// TIA Portal V20 export
// export: Created 2025-12-01T14:57:42.2360027Z, ExportSetting None, DisplayName Totally Integrated Automation Portal, DisplayVersion V20 Update 3, DisplayName TIA Portal Openness, DisplayVersion V20 Update 3, DisplayName TIA Portal Version Control Interface, DisplayVersion V20 Update 3, DisplayName STEP 7 Professional, DisplayVersion V20 Update 3, DisplayName STEP 7 Safety, DisplayVersion V20 Update 2, DisplayName WinCC Basic/Comfort/Advanced, DisplayVersion V20 Update 3, DisplayName WinCC Professional, DisplayVersion V20 Update 3, DisplayName WinCC Unified, DisplayVersion V20 Update 3
FUNCTION_BLOCK "FB383_GarrasLenze_Paletizador_NDD_E3S3"   // FB383, LAD
{ S7_Optimized_Access := 'FALSE' }
// stored: AutoNumber false, SetENOAutomatically false
   VAR_INPUT
      Mesa : UInt;   // Mesa de la FB
      NDB_ConfigNDD : UInt;
      NDB_DatosNDD : UInt;   // DB de Configuracion Particular del NDD
      OffsetDatosGarra : UInt;
      DesHabilitar_Garra : Bool;
      Mantenimiento : Bool;
      Error_Tx : Bool;
      EnTension : Bool;   // Existe Tension en la Mesa
      TermicoFRENO_Garra : Bool;
      Garra_PresCarga : Bool;
      EM_Garra_Down : Bool;
      Garra_Down : Bool;
      Garra_FinPaletizado : Bool;
      Garra_InicioPaletizado : Bool;
      EM_Garra_Up : Bool;
      P_Puesto_Capa : Bool;
      P_Puesto_Subir : Bool;
      P_Puesto_Bajar : Bool;
      BarreraNivel : Bool;
      F_EnvMens_PMx : Bool;
      Manual_GarraUp : Bool;
      Manual_GarraDown : Bool;
      Homming_Garra : Bool;   // Realizar el Homing del Variador de la Horquilla (RefCero >> Out)
      pHsRef_Garra : Bool;
      V_TOut_MovGarra : Time;
   END_VAR
   VAR_OUTPUT
      P_EnvMens_PMx : Bool;
   END_VAR
   VAR_IN_OUT
      Interlock_Garras : "NDD_Interlock_Garras";
   END_VAR
   VAR
      TOut_MovGarras { S7_SetPoint := 'True'} : TON_TIME;
      TEstableMovGarras { S7_SetPoint := 'True'} : TON_TIME;
      TEsperaMoverGarras { S7_SetPoint := 'True'} : TON_TIME;
      MemoAlturaPedido : Int;
      MemoEventoPaletizado : UInt;
      MemoPosicionAcutual_Garras : Int;
      PosicionActual_Garras : Int;
      PosicionUp_Garras : Int;
      PosicionDown_Garras : Int;
      PosicionMover_Garras : Int;
      ConsignaFR_Garras : Int;
      SubjectArea_Garras : Word;
      IDArea_Garras : Word;
      NodoNoPres_VarGarras : Bool;   // Nodo del Variador de la Horquilla - No presente
      MoverGarras : Bool;
      FinMoverGarras : Bool;
      MemoFinMoverGarras : Bool;
      PosGarrasUp_OK : Bool;
      PosGarrasDown_OK : Bool;
      PosGarrasTransfer_OK : Bool;
      Memo_NuevaCapa : Bool;
      MA_Puesto_NuevaCapa : Bool;
      MA_Puesto_Subir : Bool;
      MA_Puesto_Bajar : Bool;
      MA_Puesto_Baliza : Bool;
      MA_Garras_Subir : Bool;
      MA_Garras_Bajar : Bool;
      GARRA_ET00 : Bool;
      GARRA_ET01 : Bool;
      GARRA_ET02 : Bool;
      GARRA_RST01 : Bool;
      GARRA_RST02 : Bool;
      GARRA_CAR01 : Bool;
      GARRA_CAR02 : Bool;
      GARRA_CAR03 : Bool;
      GARRA_CAR04 : Bool;
      GARRA_DCAR01 : Bool;
      GARRA_DCAR02 : Bool;
      GARRA_DCAR03 : Bool;
      GARRA_DCAR04 : Bool;
      STAT_P_EnvMens_PMx : Bool;
      MemoReferenciaOK_Garra : Bool;
      ErrorVar_Garra : Bool;
      ReferenciaOK_Garra : Bool;
      MemoHoming_Garra : Bool;
      EventoInicioPaletizado : Bool;
      EventoFinalPaletizado : Bool;
      EventoAlturaPedido : Bool;
   END_VAR
   VAR_TEMP
      EstadoZona : "EstadoZona";
      EstadoVI : "EstadosMesa_GarrasLenze_Paletizador_NDD";
      NodoVar_Garra : "Status_NodosProfinet";
      Guardar_AR1 : DWord;
      Guardar_AR2 : DWord;
      P_DatosGarras : DWord;
      P_NodoVar_Garras : DWord;
      DB_ConfigNDD : Word;
      DB_DatosNDD : Word;
      NumDB_DiagProfinet : Word;
      NumNodo_VarGarras : UInt;
      ByteInicial_VarGarras : UInt;
      VeloManual_Garras : Int;
      VeloPuesto_Garras : Int;
      VeloLentaUp_Garras : Int;
      VeloRapidaUp_Garras : Int;
      PosLentaUp_Garras : Int;
      VeloLentaDown_Garras : Int;
      VeloRapidaDown_Garras : Int;
      PosLentaDown_Garras : Int;
      AuxMargen : Int;
      AuxPosMax : Int;
      AuxPosMin : Int;
      AuxAlturaPedidoMax : Int;
      AuxAlturaPedidoMin : Int;
      MargenPedido : Int;
      TempInt : Int;
      AuxEstados : Bool;
      DestinoGarra_DOWN : Bool;
      DestinoGarra_UP : Bool;
      MoverGarra_LentaDOWN : Bool;
      MoverGarra_LentaUP : Bool;
      CalcularAlturaPedido : Bool;
   END_VAR
   VAR_TEMP   // added for the SCL form of the ladder/FBD networks
      _w1 : Bool;
      _w2 : Bool;
      _w3 : Bool;
   END_VAR
BEGIN

REGION Network 1: Inicializaciones
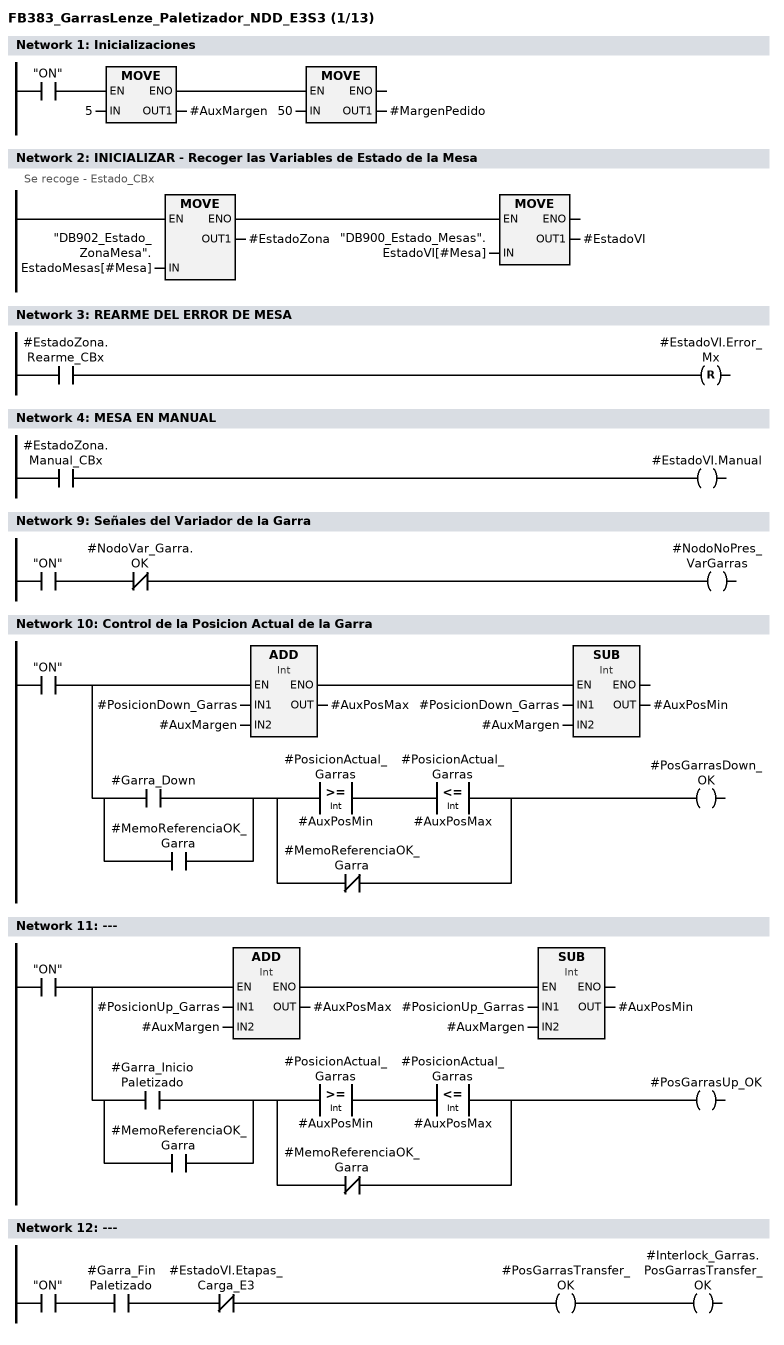
   RUNG wire#powerrail
      Contact( "ON" )
      { S7_GenerateENO := "TRUE" } Move(in := 5, out1 => #AuxMargen)
      { S7_GenerateENO := "TRUE" } Move(in := 50, out1 => #MargenPedido)
   END_RUNG
   // the same network as SCL:
   // ENO of a box is taken as its EN; it also drops when the box reports an error
   IF "ON" THEN
       #AuxMargen := 5;
       #MargenPedido := 50;
   END_IF;
END_REGION

REGION Network 2: INICIALIZAR - Recoger las Variables de Estado de la Mesa
   // Se recoge - Estado_CBx
   RUNG wire#powerrail
      Move(in := "DB902_Estado_ZonaMesa".EstadoMesas[#Mesa], out1 => #EstadoZona)
      Move(in := "DB900_Estado_Mesas".EstadoVI[#Mesa], out1 => #EstadoVI)
   END_RUNG
   // the same network as SCL:
   #EstadoZona := "DB902_Estado_ZonaMesa".EstadoMesas[#Mesa];
   #EstadoVI := "DB900_Estado_Mesas".EstadoVI[#Mesa];
END_REGION

REGION Network 3: REARME DEL ERROR DE MESA
   RUNG wire#powerrail
      Contact( #EstadoZona.Rearme_CBx )
      R_Coil( #EstadoVI.Error_Mx )
   END_RUNG
   // the same network as SCL:
   IF #EstadoZona.Rearme_CBx THEN #EstadoVI.Error_Mx := FALSE; END_IF;
END_REGION

REGION Network 4: MESA EN MANUAL
   RUNG wire#powerrail
      Contact( #EstadoZona.Manual_CBx )
      Coil( #EstadoVI.Manual )
   END_RUNG
   // the same network as SCL:
   #EstadoVI.Manual := #EstadoZona.Manual_CBx;
END_REGION

NETWORK
TITLE = Datos Internos de la Garra
// ------------------------------------------------------------------------------------
// ------------------------------------------------------------------------------------
// --- Previas

      TAR1  #Guardar_AR1;  // Guardar AR1 y AR2


// ------------------------------------------------------------------------------------
// ------------------------------------------------------------------------------------
// --- Datos iniciales

      L     #NDB_ConfigNDD;  // - DB del Config de los Paletizadores MDD
      T     #DB_ConfigNDD;  //
      L     #NDB_DatosNDD;  // - DB del Config de los Paletizadores MDD
      T     #DB_DatosNDD;

      L     #OffsetDatosGarra;  //   Puntero a los Datos de Garra
      SLD   3;
      T     #P_DatosGarras;


/////////////////////////////////////////////////////////////////////////////
/////////////////////////////////////////////////////////////////////////////
// --- Sistema de Profinet

      LAR1  P#0.0;  // - Leer Datos de los Variadores
      OPN   DB [#DB_DatosNDD];  //   del NDD

      L     DBW [AR1, P#0.0];  // - Num DB de Profinet
      T     #NumDB_DiagProfinet;
      L     DBW [AR1, P#8.0];  // - Nodos de los Variadores
      T     #NumNodo_VarGarras;
      L     DBW [AR1, P#14.0];  // - Direcciones de los Variadores
      T     #ByteInicial_VarGarras;

      L     P##NodoVar_Garra;  // Puntero del Estado del Nodo del Variador de Garra (TEMPORAL)
      T     #P_NodoVar_Garras;



NETWORK
TITLE = ----
// ------------------------------------------------------------------------------------
// ------------------------------------------------------------------------------------
// --- Datos Generales de Configuracion de los NDD

      LAR1  P#0.0;  // - Leer Datos de Velocidad de la Garra
      OPN   DB [#DB_ConfigNDD];

      L     DBW [AR1, P#30.0];  // - Velocidad en Manual
      T     #VeloManual_Garras;
      L     DBW [AR1, P#32.0];  // - Velocidad en el Puesto
      T     #VeloPuesto_Garras;

      L     DBW [AR1, P#34.0];  // - Velocidad en Auto Up
      T     #VeloLentaUp_Garras;
      L     DBW [AR1, P#36.0];
      T     #VeloRapidaUp_Garras;

      L     DBW [AR1, P#38.0];  // - Velocidad en Auto Down
      T     #VeloLentaDown_Garras;
      L     DBW [AR1, P#40.0];
      T     #VeloRapidaDown_Garras;

      L     DBW [AR1, P#42.0];  // - Posiciones para Cambio de Velocidad
      T     #PosLentaUp_Garras;
      L     DBW [AR1, P#44.0];
      T     #PosLentaDown_Garras;



NETWORK
TITLE = ----
// ------------------------------------------------------------------------------------
// ------------------------------------------------------------------------------------
// --- Datos Particulares de la Garra del NDD

      LAR1  #P_DatosGarras;  // - Leer Datos de la Garra
      OPN   DB [#DB_DatosNDD];
      L     DBD [AR1, P#0.0];
      T     #PosicionUp_Garras;
      L     DBD [AR1, P#4.0];
      T     #PosicionDown_Garras;


// ------------------------------------------------------------------------------------
// ------------------------------------------------------------------------------------
// --- Estado del Nodo de PROFINET del Variador de la Garra (DANFFOS)

      L     #NumNodo_VarGarras;  // Nodo de Profinet
      L     1;
      -I;
      L     2;  // Longitud registro datos
      *I;
      SLD   3;
      LAR1;

      OPN   DB [#NumDB_DiagProfinet];  // Leer estado del Nodo de PROFINET
      L     DBW [AR1, P#0.0];
      T     LW [#P_NodoVar_Garras];



NETWORK
TITLE = ---
// ------------------------------------------------------------------------------------
// ------------------------------------------------------------------------------------
// --- Final de Datos Inicialies

      LAR1  #Guardar_AR1;  // Recuperar AR1 y AR2



REGION Network 9: Señales del Variador de la Garra
   RUNG wire#powerrail
      Contact( "ON" )
      I_Contact( #NodoVar_Garra.OK )
      Coil( #NodoNoPres_VarGarras )
   END_RUNG
   // the same network as SCL:
   #NodoNoPres_VarGarras := "ON" AND NOT #NodoVar_Garra.OK;
END_REGION

REGION Network 10: Control de la Posicion Actual de la Garra
   RUNG wire#powerrail
      Contact( "ON" )
      wire#w1
      { S7_Templates := "SrcType := Int"; S7_GenerateENO := "TRUE" } Add(in1 := #PosicionDown_Garras, in2 := #AuxMargen, out => #AuxPosMax)
      { S7_Templates := "SrcType := Int"; S7_GenerateENO := "TRUE" } Sub(in1 := #PosicionDown_Garras, in2 := #AuxMargen, out => #AuxPosMin)
   END_RUNG
   RUNG wire#w1
      Contact( #Garra_Down )
      wire#w2
      { S7_Templates := "SrcType := Int" } GE_Contact(in1 := #PosicionActual_Garras, in2 := #AuxPosMin)
      { S7_Templates := "SrcType := Int" } LE_Contact(in1 := #PosicionActual_Garras, in2 := #AuxPosMax)
      wire#w3
      Coil( #PosGarrasDown_OK )
   END_RUNG
   RUNG wire#w1
      Contact( #MemoReferenciaOK_Garra )
   END_RUNG wire#w2
   RUNG wire#w2
      I_Contact( #MemoReferenciaOK_Garra )
   END_RUNG wire#w3
   // the same network as SCL:
   // ENO of a box is taken as its EN; it also drops when the box reports an error
   IF "ON" THEN
       #AuxPosMax := #PosicionDown_Garras + #AuxMargen;
       #AuxPosMin := #PosicionDown_Garras - #AuxMargen;
   END_IF;
   #PosGarrasDown_OK := "ON" AND (#Garra_Down OR #MemoReferenciaOK_Garra) AND (((#PosicionActual_Garras >= #AuxPosMin) AND (#PosicionActual_Garras <= #AuxPosMax)) OR NOT #MemoReferenciaOK_Garra);
END_REGION

REGION Network 11: ---
   RUNG wire#powerrail
      Contact( "ON" )
      wire#w1
      { S7_Templates := "SrcType := Int"; S7_GenerateENO := "TRUE" } Add(in1 := #PosicionUp_Garras, in2 := #AuxMargen, out => #AuxPosMax)
      { S7_Templates := "SrcType := Int"; S7_GenerateENO := "TRUE" } Sub(in1 := #PosicionUp_Garras, in2 := #AuxMargen, out => #AuxPosMin)
   END_RUNG
   RUNG wire#w1
      Contact( #Garra_InicioPaletizado )
      wire#w2
      { S7_Templates := "SrcType := Int" } GE_Contact(in1 := #PosicionActual_Garras, in2 := #AuxPosMin)
      { S7_Templates := "SrcType := Int" } LE_Contact(in1 := #PosicionActual_Garras, in2 := #AuxPosMax)
      wire#w3
      Coil( #PosGarrasUp_OK )
   END_RUNG
   RUNG wire#w1
      Contact( #MemoReferenciaOK_Garra )
   END_RUNG wire#w2
   RUNG wire#w2
      I_Contact( #MemoReferenciaOK_Garra )
   END_RUNG wire#w3
   // the same network as SCL:
   // ENO of a box is taken as its EN; it also drops when the box reports an error
   IF "ON" THEN
       #AuxPosMax := #PosicionUp_Garras + #AuxMargen;
       #AuxPosMin := #PosicionUp_Garras - #AuxMargen;
   END_IF;
   #PosGarrasUp_OK := "ON" AND (#Garra_InicioPaletizado OR #MemoReferenciaOK_Garra) AND (((#PosicionActual_Garras >= #AuxPosMin) AND (#PosicionActual_Garras <= #AuxPosMax)) OR NOT #MemoReferenciaOK_Garra);
END_REGION

REGION Network 12: ---
   RUNG wire#powerrail
      Contact( "ON" )
      Contact( #Garra_FinPaletizado )
      I_Contact( #EstadoVI.Etapas_Carga_E3 )
      Coil( #PosGarrasTransfer_OK )
      Coil( #Interlock_Garras.PosGarrasTransfer_OK )
   END_RUNG
   // the same network as SCL:
   #PosGarrasTransfer_OK := "ON" AND #Garra_FinPaletizado AND NOT #EstadoVI.Etapas_Carga_E3;
   #Interlock_Garras.PosGarrasTransfer_OK := #PosGarrasTransfer_OK;
END_REGION

REGION Network 13: ----
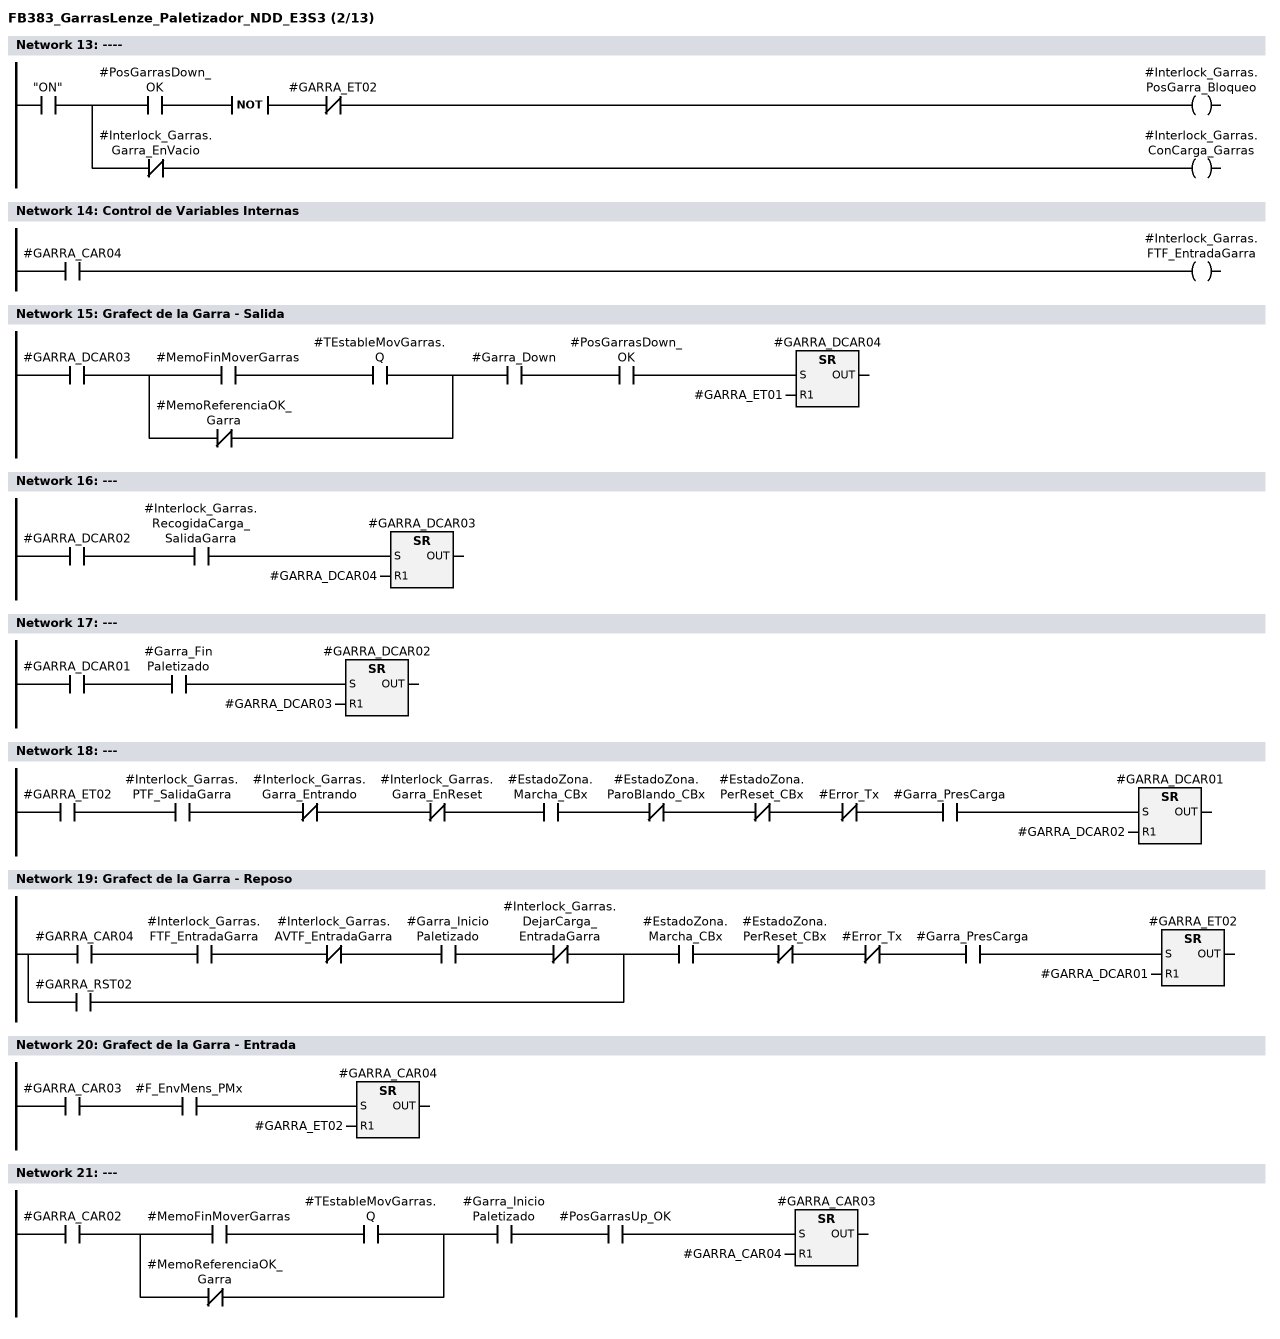
   RUNG wire#powerrail
      Contact( "ON" )
      wire#w1
      Contact( #PosGarrasDown_OK )
      Not()
      I_Contact( #GARRA_ET02 )
      Coil( #Interlock_Garras.PosGarra_Bloqueo )
   END_RUNG
   RUNG wire#w1
      I_Contact( #Interlock_Garras.Garra_EnVacio )
      Coil( #Interlock_Garras.ConCarga_Garras )
   END_RUNG
   // the same network as SCL:
   #Interlock_Garras.PosGarra_Bloqueo := NOT ("ON" AND #PosGarrasDown_OK) AND NOT #GARRA_ET02;
   #Interlock_Garras.ConCarga_Garras := "ON" AND NOT #Interlock_Garras.Garra_EnVacio;
END_REGION

REGION Network 14: Control de Variables Internas
   RUNG wire#powerrail
      Contact( #GARRA_CAR04 )
      Coil( #Interlock_Garras.FTF_EntradaGarra )
   END_RUNG
   // the same network as SCL:
   #Interlock_Garras.FTF_EntradaGarra := #GARRA_CAR04;
END_REGION

REGION Network 15: Grafect de la Garra - Salida
   RUNG wire#powerrail
      Contact( #GARRA_DCAR03 )
      wire#w1
      Contact( #MemoFinMoverGarras )
      Contact( #TEstableMovGarras.Q )
      wire#w2
      Contact( #Garra_Down )
      Contact( #PosGarrasDown_OK )
      S_SR(operand := #GARRA_DCAR04, r1 := #GARRA_ET01)
   END_RUNG
   RUNG wire#w1
      I_Contact( #MemoReferenciaOK_Garra )
   END_RUNG wire#w2
   // the same network as SCL:
   IF #GARRA_DCAR03 AND ((#MemoFinMoverGarras AND #TEstableMovGarras.Q) OR NOT #MemoReferenciaOK_Garra) AND #Garra_Down AND #PosGarrasDown_OK THEN
       #GARRA_DCAR04 := TRUE;   // SR flip-flop
   END_IF;
   IF #GARRA_ET01 THEN #GARRA_DCAR04 := FALSE; END_IF;
END_REGION

REGION Network 16: ---
   RUNG wire#powerrail
      Contact( #GARRA_DCAR02 )
      Contact( #Interlock_Garras.RecogidaCarga_SalidaGarra )
      S_SR(operand := #GARRA_DCAR03, r1 := #GARRA_DCAR04)
   END_RUNG
   // the same network as SCL:
   IF #GARRA_DCAR02 AND #Interlock_Garras.RecogidaCarga_SalidaGarra THEN
       #GARRA_DCAR03 := TRUE;   // SR flip-flop
   END_IF;
   IF #GARRA_DCAR04 THEN #GARRA_DCAR03 := FALSE; END_IF;
END_REGION

REGION Network 17: ---
   RUNG wire#powerrail
      Contact( #GARRA_DCAR01 )
      Contact( #Garra_FinPaletizado )
      S_SR(operand := #GARRA_DCAR02, r1 := #GARRA_DCAR03)
   END_RUNG
   // the same network as SCL:
   IF #GARRA_DCAR01 AND #Garra_FinPaletizado THEN
       #GARRA_DCAR02 := TRUE;   // SR flip-flop
   END_IF;
   IF #GARRA_DCAR03 THEN #GARRA_DCAR02 := FALSE; END_IF;
END_REGION

REGION Network 18: ---
   RUNG wire#powerrail
      Contact( #GARRA_ET02 )
      Contact( #Interlock_Garras.PTF_SalidaGarra )
      I_Contact( #Interlock_Garras.Garra_Entrando )
      I_Contact( #Interlock_Garras.Garra_EnReset )
      Contact( #EstadoZona.Marcha_CBx )
      I_Contact( #EstadoZona.ParoBlando_CBx )
      I_Contact( #EstadoZona.PerReset_CBx )
      I_Contact( #Error_Tx )
      Contact( #Garra_PresCarga )
      S_SR(operand := #GARRA_DCAR01, r1 := #GARRA_DCAR02)
   END_RUNG
   // the same network as SCL:
   IF #GARRA_ET02 AND #Interlock_Garras.PTF_SalidaGarra AND NOT #Interlock_Garras.Garra_Entrando AND NOT #Interlock_Garras.Garra_EnReset AND #EstadoZona.Marcha_CBx AND NOT #EstadoZona.ParoBlando_CBx AND NOT #EstadoZona.PerReset_CBx AND NOT #Error_Tx AND #Garra_PresCarga THEN
       #GARRA_DCAR01 := TRUE;   // SR flip-flop
   END_IF;
   IF #GARRA_DCAR02 THEN #GARRA_DCAR01 := FALSE; END_IF;
END_REGION

REGION Network 19: Grafect de la Garra - Reposo
   RUNG wire#powerrail
      Contact( #GARRA_CAR04 )
      Contact( #Interlock_Garras.FTF_EntradaGarra )
      I_Contact( #Interlock_Garras.AVTF_EntradaGarra )
      Contact( #Garra_InicioPaletizado )
      I_Contact( #Interlock_Garras.DejarCarga_EntradaGarra )
      wire#w1
      Contact( #EstadoZona.Marcha_CBx )
      I_Contact( #EstadoZona.PerReset_CBx )
      I_Contact( #Error_Tx )
      Contact( #Garra_PresCarga )
      S_SR(operand := #GARRA_ET02, r1 := #GARRA_DCAR01)
   END_RUNG
   RUNG wire#powerrail
      Contact( #GARRA_RST02 )
   END_RUNG wire#w1
   // the same network as SCL:
   IF ((#GARRA_CAR04 AND #Interlock_Garras.FTF_EntradaGarra AND NOT #Interlock_Garras.AVTF_EntradaGarra AND #Garra_InicioPaletizado AND NOT #Interlock_Garras.DejarCarga_EntradaGarra) OR #GARRA_RST02) AND #EstadoZona.Marcha_CBx AND NOT #EstadoZona.PerReset_CBx AND NOT #Error_Tx AND #Garra_PresCarga THEN
       #GARRA_ET02 := TRUE;   // SR flip-flop
   END_IF;
   IF #GARRA_DCAR01 THEN #GARRA_ET02 := FALSE; END_IF;
END_REGION

REGION Network 20: Grafect de la Garra - Entrada
   RUNG wire#powerrail
      Contact( #GARRA_CAR03 )
      Contact( #F_EnvMens_PMx )
      S_SR(operand := #GARRA_CAR04, r1 := #GARRA_ET02)
   END_RUNG
   // the same network as SCL:
   IF #GARRA_CAR03 AND #F_EnvMens_PMx THEN
       #GARRA_CAR04 := TRUE;   // SR flip-flop
   END_IF;
   IF #GARRA_ET02 THEN #GARRA_CAR04 := FALSE; END_IF;
END_REGION

REGION Network 21: ---
   RUNG wire#powerrail
      Contact( #GARRA_CAR02 )
      wire#w1
      Contact( #MemoFinMoverGarras )
      Contact( #TEstableMovGarras.Q )
      wire#w2
      Contact( #Garra_InicioPaletizado )
      Contact( #PosGarrasUp_OK )
      S_SR(operand := #GARRA_CAR03, r1 := #GARRA_CAR04)
   END_RUNG
   RUNG wire#w1
      I_Contact( #MemoReferenciaOK_Garra )
   END_RUNG wire#w2
   // the same network as SCL:
   IF #GARRA_CAR02 AND ((#MemoFinMoverGarras AND #TEstableMovGarras.Q) OR NOT #MemoReferenciaOK_Garra) AND #Garra_InicioPaletizado AND #PosGarrasUp_OK THEN
       #GARRA_CAR03 := TRUE;   // SR flip-flop
   END_IF;
   IF #GARRA_CAR04 THEN #GARRA_CAR03 := FALSE; END_IF;
END_REGION

REGION Network 22: ---
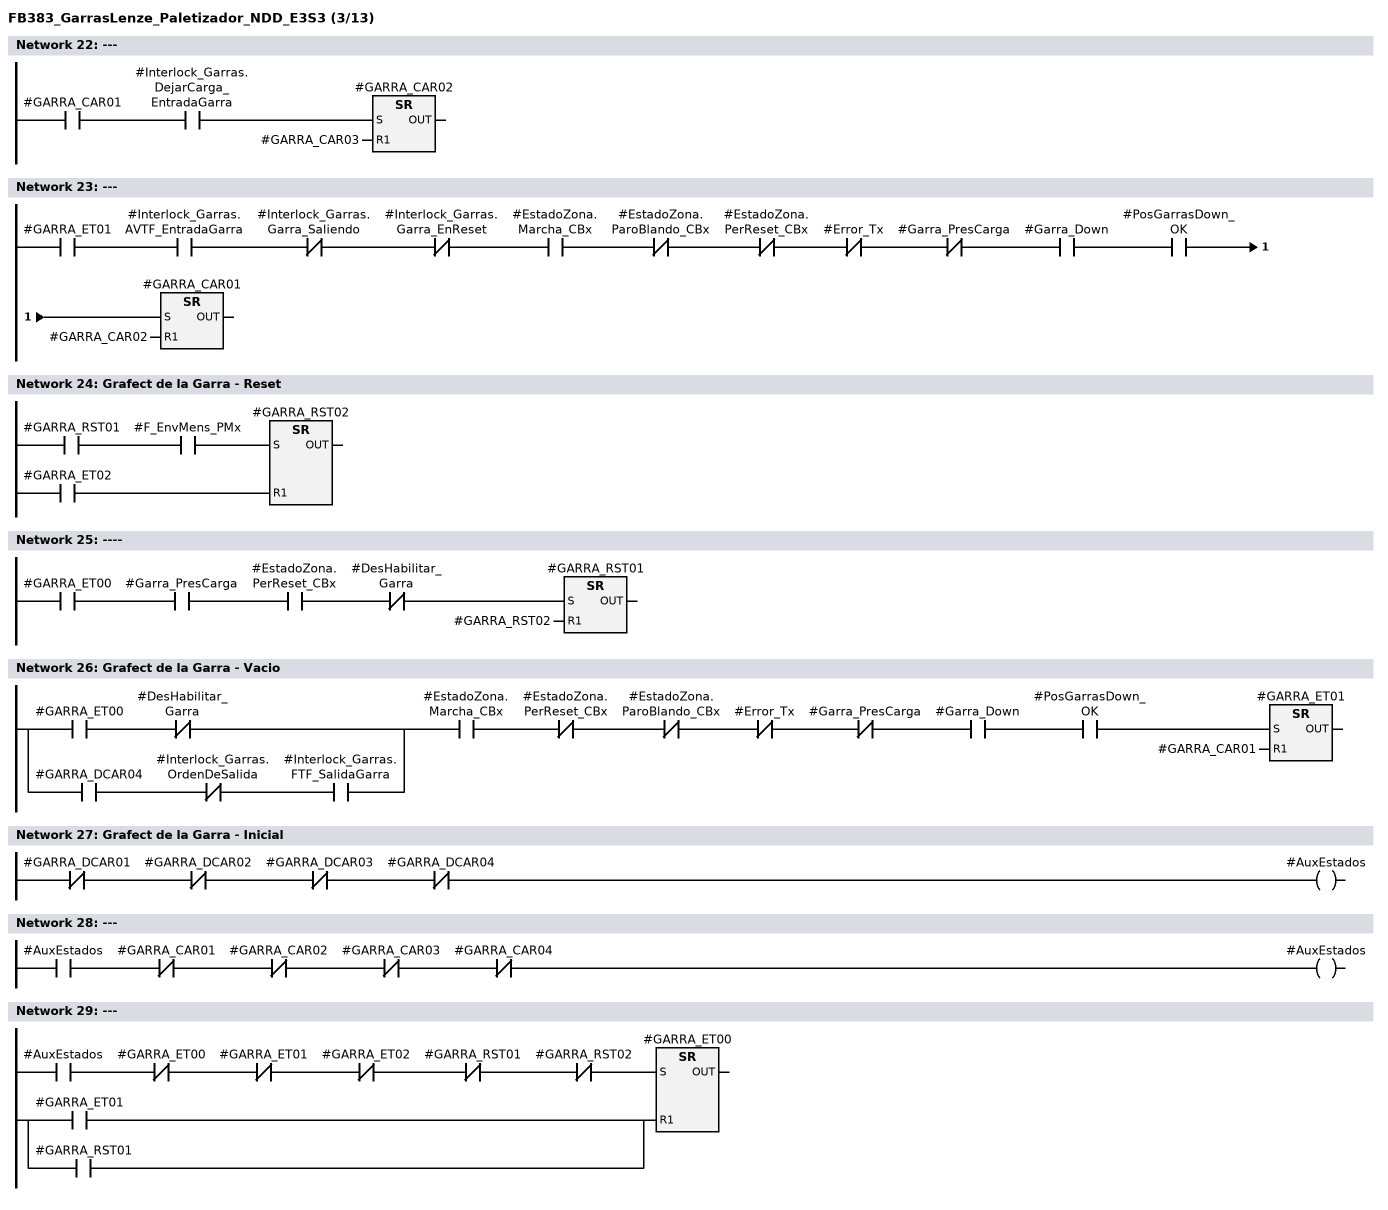
   RUNG wire#powerrail
      Contact( #GARRA_CAR01 )
      Contact( #Interlock_Garras.DejarCarga_EntradaGarra )
      S_SR(operand := #GARRA_CAR02, r1 := #GARRA_CAR03)
   END_RUNG
   // the same network as SCL:
   IF #GARRA_CAR01 AND #Interlock_Garras.DejarCarga_EntradaGarra THEN
       #GARRA_CAR02 := TRUE;   // SR flip-flop
   END_IF;
   IF #GARRA_CAR03 THEN #GARRA_CAR02 := FALSE; END_IF;
END_REGION

REGION Network 23: ---
   RUNG wire#powerrail
      Contact( #GARRA_ET01 )
      Contact( #Interlock_Garras.AVTF_EntradaGarra )
      I_Contact( #Interlock_Garras.Garra_Saliendo )
      I_Contact( #Interlock_Garras.Garra_EnReset )
      Contact( #EstadoZona.Marcha_CBx )
      I_Contact( #EstadoZona.ParoBlando_CBx )
      I_Contact( #EstadoZona.PerReset_CBx )
      I_Contact( #Error_Tx )
      I_Contact( #Garra_PresCarga )
      Contact( #Garra_Down )
      Contact( #PosGarrasDown_OK )
      S_SR(operand := #GARRA_CAR01, r1 := #GARRA_CAR02)
   END_RUNG
   // the same network as SCL:
   IF #GARRA_ET01 AND #Interlock_Garras.AVTF_EntradaGarra AND NOT #Interlock_Garras.Garra_Saliendo AND NOT #Interlock_Garras.Garra_EnReset AND #EstadoZona.Marcha_CBx AND NOT #EstadoZona.ParoBlando_CBx AND NOT #EstadoZona.PerReset_CBx AND NOT #Error_Tx AND NOT #Garra_PresCarga AND #Garra_Down AND #PosGarrasDown_OK THEN
       #GARRA_CAR01 := TRUE;   // SR flip-flop
   END_IF;
   IF #GARRA_CAR02 THEN #GARRA_CAR01 := FALSE; END_IF;
END_REGION

REGION Network 24: Grafect de la Garra - Reset
   RUNG wire#powerrail
      Contact( #GARRA_RST01 )
      Contact( #F_EnvMens_PMx )
      S_SR(operand := #GARRA_RST02, r1 := wire#w1)
   END_RUNG
   RUNG wire#powerrail
      Contact( #GARRA_ET02 )
   END_RUNG wire#w1
   // the same network as SCL:
   IF #GARRA_RST01 AND #F_EnvMens_PMx THEN
       #GARRA_RST02 := TRUE;   // SR flip-flop
   END_IF;
   IF #GARRA_ET02 THEN #GARRA_RST02 := FALSE; END_IF;
END_REGION

REGION Network 25: ----
   RUNG wire#powerrail
      Contact( #GARRA_ET00 )
      Contact( #Garra_PresCarga )
      Contact( #EstadoZona.PerReset_CBx )
      I_Contact( #DesHabilitar_Garra )
      S_SR(operand := #GARRA_RST01, r1 := #GARRA_RST02)
   END_RUNG
   // the same network as SCL:
   IF #GARRA_ET00 AND #Garra_PresCarga AND #EstadoZona.PerReset_CBx AND NOT #DesHabilitar_Garra THEN
       #GARRA_RST01 := TRUE;   // SR flip-flop
   END_IF;
   IF #GARRA_RST02 THEN #GARRA_RST01 := FALSE; END_IF;
END_REGION

REGION Network 26: Grafect de la Garra - Vacio
   RUNG wire#powerrail
      Contact( #GARRA_ET00 )
      I_Contact( #DesHabilitar_Garra )
      wire#w1
      Contact( #EstadoZona.Marcha_CBx )
      I_Contact( #EstadoZona.PerReset_CBx )
      I_Contact( #EstadoZona.ParoBlando_CBx )
      I_Contact( #Error_Tx )
      I_Contact( #Garra_PresCarga )
      Contact( #Garra_Down )
      Contact( #PosGarrasDown_OK )
      S_SR(operand := #GARRA_ET01, r1 := #GARRA_CAR01)
   END_RUNG
   RUNG wire#powerrail
      Contact( #GARRA_DCAR04 )
      I_Contact( #Interlock_Garras.OrdenDeSalida )
      Contact( #Interlock_Garras.FTF_SalidaGarra )
   END_RUNG wire#w1
   // the same network as SCL:
   IF ((#GARRA_ET00 AND NOT #DesHabilitar_Garra) OR (#GARRA_DCAR04 AND NOT #Interlock_Garras.OrdenDeSalida AND #Interlock_Garras.FTF_SalidaGarra)) AND #EstadoZona.Marcha_CBx AND NOT #EstadoZona.PerReset_CBx AND NOT #EstadoZona.ParoBlando_CBx AND NOT #Error_Tx AND NOT #Garra_PresCarga AND #Garra_Down AND #PosGarrasDown_OK THEN
       #GARRA_ET01 := TRUE;   // SR flip-flop
   END_IF;
   IF #GARRA_CAR01 THEN #GARRA_ET01 := FALSE; END_IF;
END_REGION

REGION Network 27: Grafect de la Garra - Inicial
   RUNG wire#powerrail
      I_Contact( #GARRA_DCAR01 )
      I_Contact( #GARRA_DCAR02 )
      I_Contact( #GARRA_DCAR03 )
      I_Contact( #GARRA_DCAR04 )
      Coil( #AuxEstados )
   END_RUNG
   // the same network as SCL:
   #AuxEstados := NOT #GARRA_DCAR01 AND NOT #GARRA_DCAR02 AND NOT #GARRA_DCAR03 AND NOT #GARRA_DCAR04;
END_REGION

REGION Network 28: ---
   RUNG wire#powerrail
      Contact( #AuxEstados )
      I_Contact( #GARRA_CAR01 )
      I_Contact( #GARRA_CAR02 )
      I_Contact( #GARRA_CAR03 )
      I_Contact( #GARRA_CAR04 )
      Coil( #AuxEstados )
   END_RUNG
   // the same network as SCL:
   #AuxEstados := #AuxEstados AND NOT #GARRA_CAR01 AND NOT #GARRA_CAR02 AND NOT #GARRA_CAR03 AND NOT #GARRA_CAR04;
END_REGION

REGION Network 29: ---
   RUNG wire#powerrail
      Contact( #AuxEstados )
      I_Contact( #GARRA_ET00 )
      I_Contact( #GARRA_ET01 )
      I_Contact( #GARRA_ET02 )
      I_Contact( #GARRA_RST01 )
      I_Contact( #GARRA_RST02 )
      S_SR(operand := #GARRA_ET00, r1 := wire#w1)
   END_RUNG
   RUNG wire#powerrail
      Contact( #GARRA_ET01 )
   END_RUNG wire#w1
   RUNG wire#powerrail
      Contact( #GARRA_RST01 )
   END_RUNG wire#w1
   // the same network as SCL:
   IF #AuxEstados AND NOT #GARRA_ET00 AND NOT #GARRA_ET01 AND NOT #GARRA_ET02 AND NOT #GARRA_RST01 AND NOT #GARRA_RST02 THEN
       #GARRA_ET00 := TRUE;   // SR flip-flop
   END_IF;
   IF #GARRA_ET01 OR #GARRA_RST01 THEN #GARRA_ET00 := FALSE; END_IF;
END_REGION

REGION Network 30: Fin Reset y Fin Paro Blando
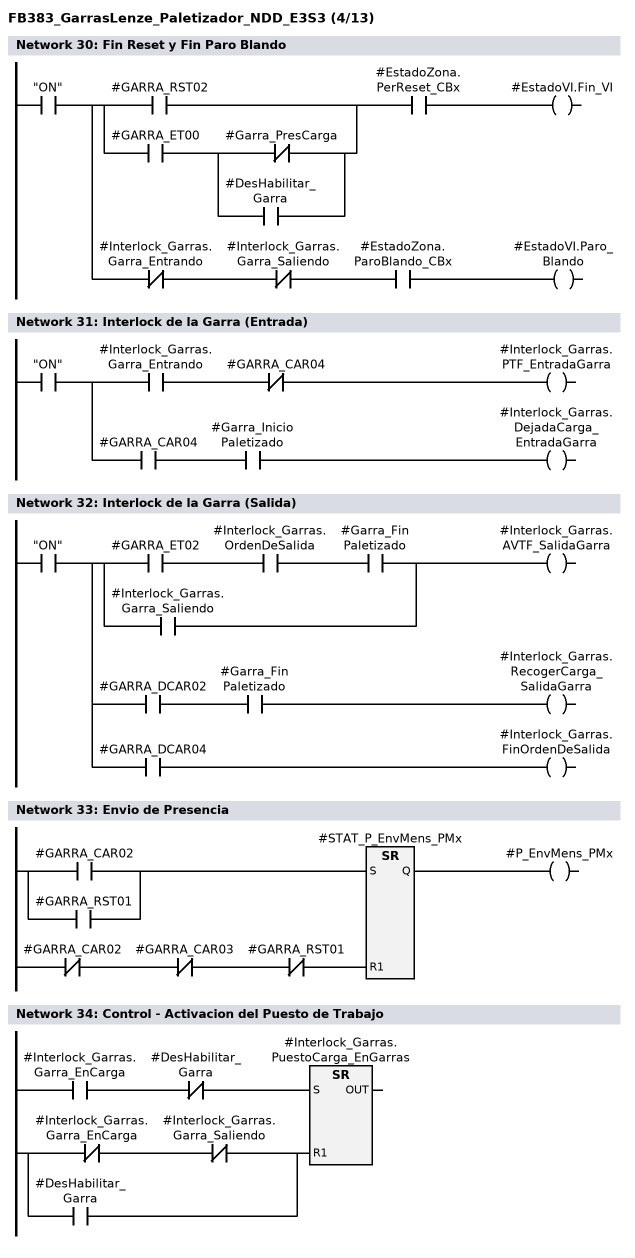
   RUNG wire#powerrail
      Contact( "ON" )
      wire#w1
      Contact( #GARRA_RST02 )
      wire#w2
      Contact( #EstadoZona.PerReset_CBx )
      Coil( #EstadoVI.Fin_VI )
   END_RUNG
   RUNG wire#w1
      Contact( #GARRA_ET00 )
      wire#w3
      I_Contact( #Garra_PresCarga )
   END_RUNG wire#w2
   RUNG wire#w3
      Contact( #DesHabilitar_Garra )
   END_RUNG wire#w2
   RUNG wire#w1
      I_Contact( #Interlock_Garras.Garra_Entrando )
      I_Contact( #Interlock_Garras.Garra_Saliendo )
      Contact( #EstadoZona.ParoBlando_CBx )
      Coil( #EstadoVI.Paro_Blando )
   END_RUNG
   // the same network as SCL:
   #EstadoVI.Fin_VI := "ON" AND (#GARRA_RST02 OR (#GARRA_ET00 AND (NOT #Garra_PresCarga OR #DesHabilitar_Garra))) AND #EstadoZona.PerReset_CBx;
   #EstadoVI.Paro_Blando := "ON" AND NOT #Interlock_Garras.Garra_Entrando AND NOT #Interlock_Garras.Garra_Saliendo AND #EstadoZona.ParoBlando_CBx;
END_REGION

REGION Network 31: Interlock de la Garra (Entrada)
   RUNG wire#powerrail
      Contact( "ON" )
      wire#w1
      Contact( #Interlock_Garras.Garra_Entrando )
      I_Contact( #GARRA_CAR04 )
      Coil( #Interlock_Garras.PTF_EntradaGarra )
   END_RUNG
   RUNG wire#w1
      Contact( #GARRA_CAR04 )
      Contact( #Garra_InicioPaletizado )
      Coil( #Interlock_Garras.DejadaCarga_EntradaGarra )
   END_RUNG
   // the same network as SCL:
   #Interlock_Garras.PTF_EntradaGarra := "ON" AND #Interlock_Garras.Garra_Entrando AND NOT #GARRA_CAR04;
   #Interlock_Garras.DejadaCarga_EntradaGarra := "ON" AND #GARRA_CAR04 AND #Garra_InicioPaletizado;
END_REGION

REGION Network 32: Interlock de la Garra (Salida)
   RUNG wire#powerrail
      Contact( "ON" )
      wire#w1
      Contact( #GARRA_ET02 )
      Contact( #Interlock_Garras.OrdenDeSalida )
      Contact( #Garra_FinPaletizado )
      wire#w2
      Coil( #Interlock_Garras.AVTF_SalidaGarra )
   END_RUNG
   RUNG wire#w1
      Contact( #Interlock_Garras.Garra_Saliendo )
   END_RUNG wire#w2
   RUNG wire#w1
      Contact( #GARRA_DCAR02 )
      Contact( #Garra_FinPaletizado )
      Coil( #Interlock_Garras.RecogerCarga_SalidaGarra )
   END_RUNG
   RUNG wire#w1
      Contact( #GARRA_DCAR04 )
      Coil( #Interlock_Garras.FinOrdenDeSalida )
   END_RUNG
   // the same network as SCL:
   #Interlock_Garras.AVTF_SalidaGarra := "ON" AND ((#GARRA_ET02 AND #Interlock_Garras.OrdenDeSalida AND #Garra_FinPaletizado) OR #Interlock_Garras.Garra_Saliendo);
   #Interlock_Garras.RecogerCarga_SalidaGarra := "ON" AND #GARRA_DCAR02 AND #Garra_FinPaletizado;
   #Interlock_Garras.FinOrdenDeSalida := "ON" AND #GARRA_DCAR04;
END_REGION

REGION Network 33: Envio de Presencia
   RUNG wire#powerrail
      Contact( #GARRA_CAR02 )
      wire#w1
      S_SR(operand := #STAT_P_EnvMens_PMx, r1 := wire#w2)
      Coil( #P_EnvMens_PMx )
   END_RUNG
   RUNG wire#powerrail
      Contact( #GARRA_RST01 )
   END_RUNG wire#w1
   RUNG wire#powerrail
      I_Contact( #GARRA_CAR02 )
      I_Contact( #GARRA_CAR03 )
      I_Contact( #GARRA_RST01 )
   END_RUNG wire#w2
   // the same network as SCL:
   IF #GARRA_CAR02 OR #GARRA_RST01 THEN
       #STAT_P_EnvMens_PMx := TRUE;   // SR flip-flop
   END_IF;
   IF NOT #GARRA_CAR02 AND NOT #GARRA_CAR03 AND NOT #GARRA_RST01 THEN #STAT_P_EnvMens_PMx := FALSE; END_IF;
   #P_EnvMens_PMx := #STAT_P_EnvMens_PMx;
END_REGION

REGION Network 34: Control - Activacion del Puesto de Trabajo
   RUNG wire#powerrail
      Contact( #Interlock_Garras.Garra_EnCarga )
      I_Contact( #DesHabilitar_Garra )
      S_SR(operand := #Interlock_Garras.PuestoCarga_EnGarras, r1 := wire#w1)
   END_RUNG
   RUNG wire#powerrail
      I_Contact( #Interlock_Garras.Garra_EnCarga )
      I_Contact( #Interlock_Garras.Garra_Saliendo )
   END_RUNG wire#w1
   RUNG wire#powerrail
      Contact( #DesHabilitar_Garra )
   END_RUNG wire#w1
   // the same network as SCL:
   IF #Interlock_Garras.Garra_EnCarga AND NOT #DesHabilitar_Garra THEN
       #Interlock_Garras.PuestoCarga_EnGarras := TRUE;   // SR flip-flop
   END_IF;
   IF (NOT #Interlock_Garras.Garra_EnCarga AND NOT #Interlock_Garras.Garra_Saliendo) OR #DesHabilitar_Garra THEN
       #Interlock_Garras.PuestoCarga_EnGarras := FALSE;
   END_IF;
END_REGION

REGION Network 35: Control - Activacion de Nueva Capa
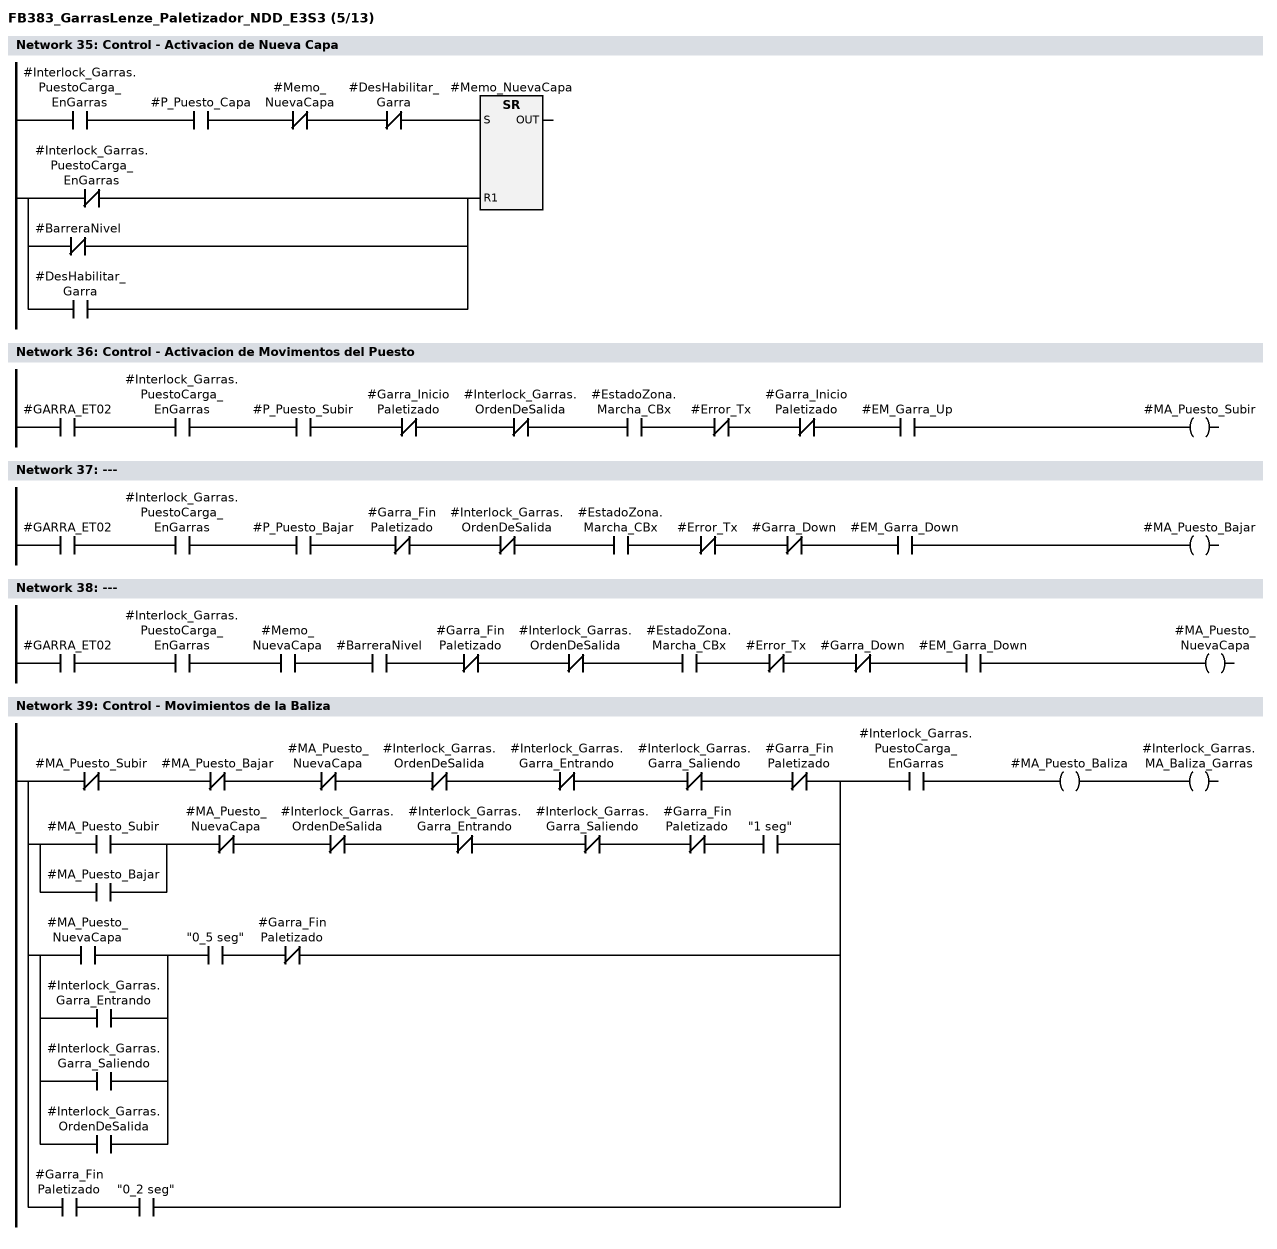
   RUNG wire#powerrail
      Contact( #Interlock_Garras.PuestoCarga_EnGarras )
      Contact( #P_Puesto_Capa )
      I_Contact( #Memo_NuevaCapa )
      I_Contact( #DesHabilitar_Garra )
      S_SR(operand := #Memo_NuevaCapa, r1 := wire#w1)
   END_RUNG
   RUNG wire#powerrail
      I_Contact( #Interlock_Garras.PuestoCarga_EnGarras )
   END_RUNG wire#w1
   RUNG wire#powerrail
      I_Contact( #BarreraNivel )
   END_RUNG wire#w1
   RUNG wire#powerrail
      Contact( #DesHabilitar_Garra )
   END_RUNG wire#w1
   // the same network as SCL:
   IF #Interlock_Garras.PuestoCarga_EnGarras AND #P_Puesto_Capa AND NOT #Memo_NuevaCapa AND NOT #DesHabilitar_Garra THEN
       #Memo_NuevaCapa := TRUE;   // SR flip-flop
   END_IF;
   IF NOT #Interlock_Garras.PuestoCarga_EnGarras OR NOT #BarreraNivel OR #DesHabilitar_Garra THEN
       #Memo_NuevaCapa := FALSE;
   END_IF;
END_REGION

REGION Network 36: Control - Activacion de Movimentos del Puesto
   RUNG wire#powerrail
      Contact( #GARRA_ET02 )
      Contact( #Interlock_Garras.PuestoCarga_EnGarras )
      Contact( #P_Puesto_Subir )
      I_Contact( #Garra_InicioPaletizado )
      I_Contact( #Interlock_Garras.OrdenDeSalida )
      Contact( #EstadoZona.Marcha_CBx )
      I_Contact( #Error_Tx )
      I_Contact( #Garra_InicioPaletizado )
      Contact( #EM_Garra_Up )
      Coil( #MA_Puesto_Subir )
   END_RUNG
   // the same network as SCL:
   #MA_Puesto_Subir := #GARRA_ET02 AND #Interlock_Garras.PuestoCarga_EnGarras AND #P_Puesto_Subir AND NOT #Garra_InicioPaletizado AND NOT #Interlock_Garras.OrdenDeSalida AND #EstadoZona.Marcha_CBx AND NOT #Error_Tx AND NOT #Garra_InicioPaletizado AND #EM_Garra_Up;
END_REGION

REGION Network 37: ---
   RUNG wire#powerrail
      Contact( #GARRA_ET02 )
      Contact( #Interlock_Garras.PuestoCarga_EnGarras )
      Contact( #P_Puesto_Bajar )
      I_Contact( #Garra_FinPaletizado )
      I_Contact( #Interlock_Garras.OrdenDeSalida )
      Contact( #EstadoZona.Marcha_CBx )
      I_Contact( #Error_Tx )
      I_Contact( #Garra_Down )
      Contact( #EM_Garra_Down )
      Coil( #MA_Puesto_Bajar )
   END_RUNG
   // the same network as SCL:
   #MA_Puesto_Bajar := #GARRA_ET02 AND #Interlock_Garras.PuestoCarga_EnGarras AND #P_Puesto_Bajar AND NOT #Garra_FinPaletizado AND NOT #Interlock_Garras.OrdenDeSalida AND #EstadoZona.Marcha_CBx AND NOT #Error_Tx AND NOT #Garra_Down AND #EM_Garra_Down;
END_REGION

REGION Network 38: ---
   RUNG wire#powerrail
      Contact( #GARRA_ET02 )
      Contact( #Interlock_Garras.PuestoCarga_EnGarras )
      Contact( #Memo_NuevaCapa )
      Contact( #BarreraNivel )
      I_Contact( #Garra_FinPaletizado )
      I_Contact( #Interlock_Garras.OrdenDeSalida )
      Contact( #EstadoZona.Marcha_CBx )
      I_Contact( #Error_Tx )
      I_Contact( #Garra_Down )
      Contact( #EM_Garra_Down )
      Coil( #MA_Puesto_NuevaCapa )
   END_RUNG
   // the same network as SCL:
   #MA_Puesto_NuevaCapa := #GARRA_ET02 AND #Interlock_Garras.PuestoCarga_EnGarras AND #Memo_NuevaCapa AND #BarreraNivel AND NOT #Garra_FinPaletizado AND NOT #Interlock_Garras.OrdenDeSalida AND #EstadoZona.Marcha_CBx AND NOT #Error_Tx AND NOT #Garra_Down AND #EM_Garra_Down;
END_REGION

REGION Network 39: Control - Movimientos de la Baliza
   RUNG wire#powerrail
      I_Contact( #MA_Puesto_Subir )
      I_Contact( #MA_Puesto_Bajar )
      I_Contact( #MA_Puesto_NuevaCapa )
      I_Contact( #Interlock_Garras.OrdenDeSalida )
      I_Contact( #Interlock_Garras.Garra_Entrando )
      I_Contact( #Interlock_Garras.Garra_Saliendo )
      I_Contact( #Garra_FinPaletizado )
      wire#w1
      Contact( #Interlock_Garras.PuestoCarga_EnGarras )
      Coil( #MA_Puesto_Baliza )
      Coil( #Interlock_Garras.MA_Baliza_Garras )
   END_RUNG
   RUNG wire#powerrail
      Contact( #MA_Puesto_Subir )
      wire#w2
      I_Contact( #MA_Puesto_NuevaCapa )
      I_Contact( #Interlock_Garras.OrdenDeSalida )
      I_Contact( #Interlock_Garras.Garra_Entrando )
      I_Contact( #Interlock_Garras.Garra_Saliendo )
      I_Contact( #Garra_FinPaletizado )
      Contact( "1 seg" )
   END_RUNG wire#w1
   RUNG wire#powerrail
      Contact( #MA_Puesto_Bajar )
   END_RUNG wire#w2
   RUNG wire#powerrail
      Contact( #MA_Puesto_NuevaCapa )
      wire#w3
      Contact( "0_5 seg" )
      I_Contact( #Garra_FinPaletizado )
   END_RUNG wire#w1
   RUNG wire#powerrail
      Contact( #Interlock_Garras.Garra_Entrando )
   END_RUNG wire#w3
   RUNG wire#powerrail
      Contact( #Interlock_Garras.Garra_Saliendo )
   END_RUNG wire#w3
   RUNG wire#powerrail
      Contact( #Interlock_Garras.OrdenDeSalida )
   END_RUNG wire#w3
   RUNG wire#powerrail
      Contact( #Garra_FinPaletizado )
      Contact( "0_2 seg" )
   END_RUNG wire#w1
   // the same network as SCL:
   #MA_Puesto_Baliza := ((NOT #MA_Puesto_Subir AND NOT #MA_Puesto_Bajar AND NOT #MA_Puesto_NuevaCapa AND NOT #Interlock_Garras.OrdenDeSalida AND NOT #Interlock_Garras.Garra_Entrando AND NOT #Interlock_Garras.Garra_Saliendo AND NOT #Garra_FinPaletizado) OR ((#MA_Puesto_Subir OR #MA_Puesto_Bajar) AND NOT #MA_Puesto_NuevaCapa AND NOT #Interlock_Garras.OrdenDeSalida AND NOT #Interlock_Garras.Garra_Entrando AND NOT #Interlock_Garras.Garra_Saliendo AND NOT #Garra_FinPaletizado AND "1 seg") OR ((#MA_Puesto_NuevaCapa OR #Interlock_Garras.Garra_Entrando OR #Interlock_Garras.Garra_Saliendo OR #Interlock_Garras.OrdenDeSalida) AND "0_5 seg" AND NOT #Garra_FinPaletizado) OR (#Garra_FinPaletizado AND "0_2 seg")) AND #Interlock_Garras.PuestoCarga_EnGarras;
   #Interlock_Garras.MA_Baliza_Garras := #MA_Puesto_Baliza;
END_REGION

REGION Network 40: Control - Movimiento de la Garra En Semi-Automatico
   // Cuidado sino tiene Referencia tambien se mueve (En Lento)
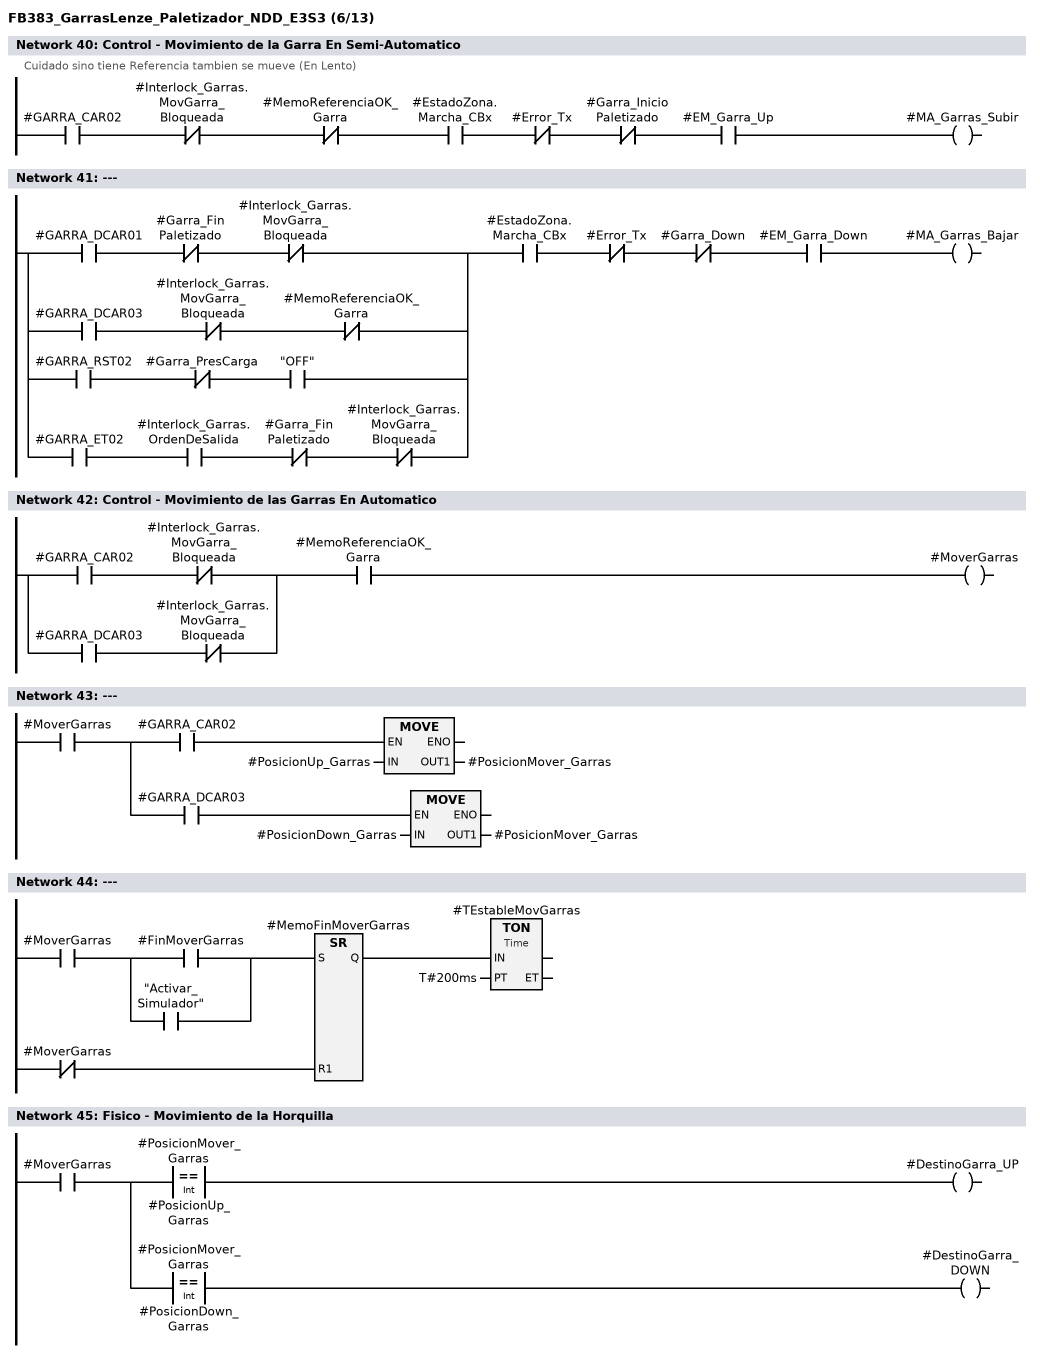
   RUNG wire#powerrail
      Contact( #GARRA_CAR02 )
      I_Contact( #Interlock_Garras.MovGarra_Bloqueada )
      I_Contact( #MemoReferenciaOK_Garra )
      Contact( #EstadoZona.Marcha_CBx )
      I_Contact( #Error_Tx )
      I_Contact( #Garra_InicioPaletizado )
      Contact( #EM_Garra_Up )
      Coil( #MA_Garras_Subir )
   END_RUNG
   // the same network as SCL:
   #MA_Garras_Subir := #GARRA_CAR02 AND NOT #Interlock_Garras.MovGarra_Bloqueada AND NOT #MemoReferenciaOK_Garra AND #EstadoZona.Marcha_CBx AND NOT #Error_Tx AND NOT #Garra_InicioPaletizado AND #EM_Garra_Up;
END_REGION

REGION Network 41: ---
   RUNG wire#powerrail
      Contact( #GARRA_DCAR01 )
      I_Contact( #Garra_FinPaletizado )
      I_Contact( #Interlock_Garras.MovGarra_Bloqueada )
      wire#w1
      Contact( #EstadoZona.Marcha_CBx )
      I_Contact( #Error_Tx )
      I_Contact( #Garra_Down )
      Contact( #EM_Garra_Down )
      Coil( #MA_Garras_Bajar )
   END_RUNG
   RUNG wire#powerrail
      Contact( #GARRA_DCAR03 )
      I_Contact( #Interlock_Garras.MovGarra_Bloqueada )
      I_Contact( #MemoReferenciaOK_Garra )
   END_RUNG wire#w1
   RUNG wire#powerrail
      Contact( #GARRA_RST02 )
      I_Contact( #Garra_PresCarga )
      Contact( "OFF" )
   END_RUNG wire#w1
   RUNG wire#powerrail
      Contact( #GARRA_ET02 )
      Contact( #Interlock_Garras.OrdenDeSalida )
      I_Contact( #Garra_FinPaletizado )
      I_Contact( #Interlock_Garras.MovGarra_Bloqueada )
   END_RUNG wire#w1
   // the same network as SCL:
   #MA_Garras_Bajar := ((#GARRA_DCAR01 AND NOT #Garra_FinPaletizado AND NOT #Interlock_Garras.MovGarra_Bloqueada) OR (#GARRA_DCAR03 AND NOT #Interlock_Garras.MovGarra_Bloqueada AND NOT #MemoReferenciaOK_Garra) OR (#GARRA_RST02 AND NOT #Garra_PresCarga AND "OFF") OR (#GARRA_ET02 AND #Interlock_Garras.OrdenDeSalida AND NOT #Garra_FinPaletizado AND NOT #Interlock_Garras.MovGarra_Bloqueada)) AND #EstadoZona.Marcha_CBx AND NOT #Error_Tx AND NOT #Garra_Down AND #EM_Garra_Down;
END_REGION

REGION Network 42: Control - Movimiento de las Garras En Automatico
   RUNG wire#powerrail
      Contact( #GARRA_CAR02 )
      I_Contact( #Interlock_Garras.MovGarra_Bloqueada )
      wire#w1
      Contact( #MemoReferenciaOK_Garra )
      Coil( #MoverGarras )
   END_RUNG
   RUNG wire#powerrail
      Contact( #GARRA_DCAR03 )
      I_Contact( #Interlock_Garras.MovGarra_Bloqueada )
   END_RUNG wire#w1
   // the same network as SCL:
   #MoverGarras := ((#GARRA_CAR02 AND NOT #Interlock_Garras.MovGarra_Bloqueada) OR (#GARRA_DCAR03 AND NOT #Interlock_Garras.MovGarra_Bloqueada)) AND #MemoReferenciaOK_Garra;
END_REGION

REGION Network 43: ---
   RUNG wire#powerrail
      Contact( #MoverGarras )
      wire#w1
      Contact( #GARRA_CAR02 )
      { S7_GenerateENO := "TRUE" } Move(in := #PosicionUp_Garras, out1 => #PosicionMover_Garras)
   END_RUNG
   RUNG wire#w1
      Contact( #GARRA_DCAR03 )
      { S7_GenerateENO := "TRUE" } Move(in := #PosicionDown_Garras, out1 => #PosicionMover_Garras)
   END_RUNG
   // the same network as SCL:
   IF #MoverGarras AND #GARRA_CAR02 THEN #PosicionMover_Garras := #PosicionUp_Garras; END_IF;
   IF #MoverGarras AND #GARRA_DCAR03 THEN #PosicionMover_Garras := #PosicionDown_Garras; END_IF;
END_REGION

REGION Network 44: ---
   RUNG wire#powerrail
      Contact( #MoverGarras )
      wire#w1
      Contact( #FinMoverGarras )
      wire#w2
      S_SR(operand := #MemoFinMoverGarras, r1 := wire#w3)
      { S7_Templates := "time_type := Time" } #TEstableMovGarras.TON(pt := T#200ms, et =>)
   END_RUNG
   RUNG wire#w1
      Contact( "Activar_Simulador" )
   END_RUNG wire#w2
   RUNG wire#powerrail
      I_Contact( #MoverGarras )
   END_RUNG wire#w3
   // the same network as SCL:
   IF #MoverGarras AND (#FinMoverGarras OR "Activar_Simulador") THEN
       #MemoFinMoverGarras := TRUE;   // SR flip-flop
   END_IF;
   IF NOT #MoverGarras THEN #MemoFinMoverGarras := FALSE; END_IF;
   #TEstableMovGarras(IN := #MemoFinMoverGarras, PT := T#200ms);   // TON
END_REGION

REGION Network 45: Fisico - Movimiento de la Horquilla
   RUNG wire#powerrail
      Contact( #MoverGarras )
      wire#w1
      { S7_Templates := "SrcType := Int" } EQ_Contact(in1 := #PosicionMover_Garras, in2 := #PosicionUp_Garras)
      Coil( #DestinoGarra_UP )
   END_RUNG
   RUNG wire#w1
      { S7_Templates := "SrcType := Int" } EQ_Contact(in1 := #PosicionMover_Garras, in2 := #PosicionDown_Garras)
      Coil( #DestinoGarra_DOWN )
   END_RUNG
   // the same network as SCL:
   #DestinoGarra_UP := #MoverGarras AND (#PosicionMover_Garras = #PosicionUp_Garras);
   #DestinoGarra_DOWN := #MoverGarras AND (#PosicionMover_Garras = #PosicionDown_Garras);
END_REGION

REGION Network 46: ---
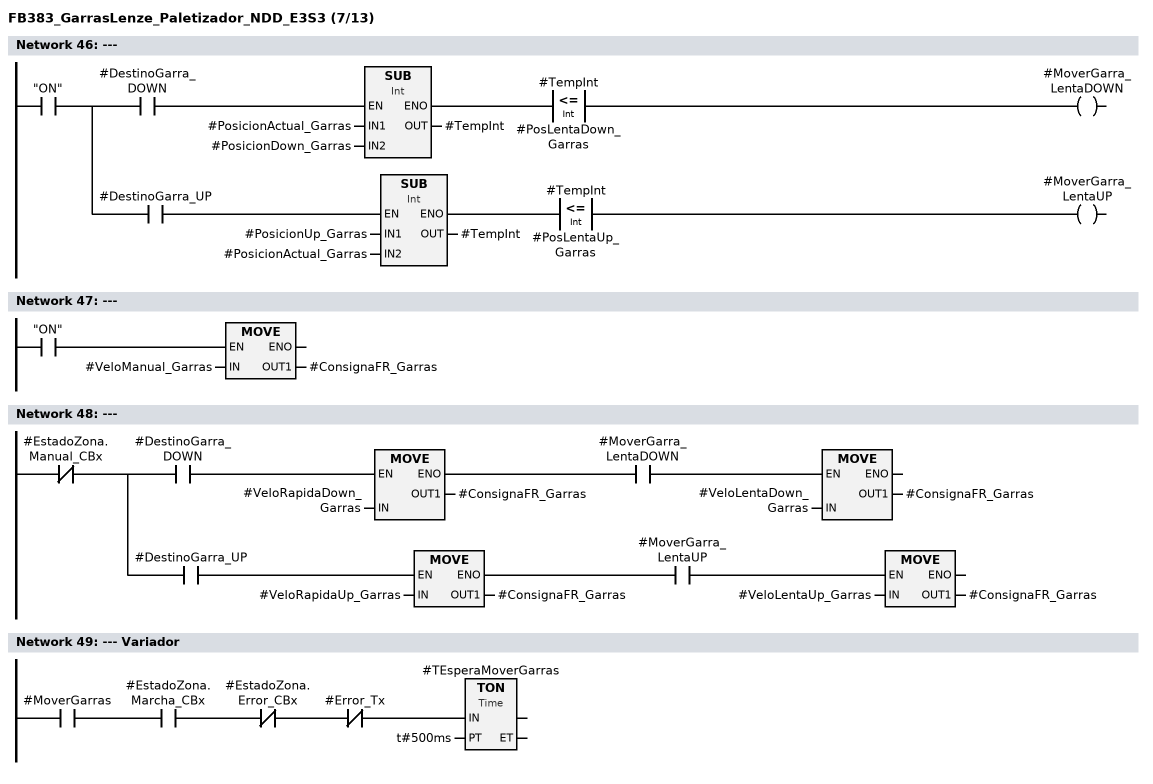
   RUNG wire#powerrail
      Contact( "ON" )
      wire#w1
      Contact( #DestinoGarra_DOWN )
      { S7_Templates := "SrcType := Int"; S7_GenerateENO := "TRUE" } Sub(in1 := #PosicionActual_Garras, in2 := #PosicionDown_Garras, out => #TempInt)
      { S7_Templates := "SrcType := Int" } LE_Contact(in1 := #TempInt, in2 := #PosLentaDown_Garras)
      Coil( #MoverGarra_LentaDOWN )
   END_RUNG
   RUNG wire#w1
      Contact( #DestinoGarra_UP )
      { S7_Templates := "SrcType := Int"; S7_GenerateENO := "TRUE" } Sub(in1 := #PosicionUp_Garras, in2 := #PosicionActual_Garras, out => #TempInt)
      { S7_Templates := "SrcType := Int" } LE_Contact(in1 := #TempInt, in2 := #PosLentaUp_Garras)
      Coil( #MoverGarra_LentaUP )
   END_RUNG
   // the same network as SCL:
   // ENO of a box is taken as its EN; it also drops when the box reports an error
   #_w1 := "ON" AND #DestinoGarra_DOWN;
   IF #_w1 THEN #TempInt := #PosicionActual_Garras - #PosicionDown_Garras; END_IF;
   #MoverGarra_LentaDOWN := #_w1 AND (#TempInt <= #PosLentaDown_Garras);
   #_w2 := "ON" AND #DestinoGarra_UP;
   IF #_w2 THEN #TempInt := #PosicionUp_Garras - #PosicionActual_Garras; END_IF;
   #MoverGarra_LentaUP := #_w2 AND (#TempInt <= #PosLentaUp_Garras);
END_REGION

REGION Network 47: ---
   RUNG wire#powerrail
      Contact( "ON" )
      { S7_GenerateENO := "TRUE" } Move(in := #VeloManual_Garras, out1 => #ConsignaFR_Garras)
   END_RUNG
   // the same network as SCL:
   IF "ON" THEN #ConsignaFR_Garras := #VeloManual_Garras; END_IF;
END_REGION

REGION Network 48: ---
   RUNG wire#powerrail
      I_Contact( #EstadoZona.Manual_CBx )
      wire#w1
      Contact( #DestinoGarra_DOWN )
      { S7_GenerateENO := "TRUE" } Move(in := #VeloRapidaDown_Garras, out1 => #ConsignaFR_Garras)
      Contact( #MoverGarra_LentaDOWN )
      { S7_GenerateENO := "TRUE" } Move(in := #VeloLentaDown_Garras, out1 => #ConsignaFR_Garras)
   END_RUNG
   RUNG wire#w1
      Contact( #DestinoGarra_UP )
      { S7_GenerateENO := "TRUE" } Move(in := #VeloRapidaUp_Garras, out1 => #ConsignaFR_Garras)
      Contact( #MoverGarra_LentaUP )
      { S7_GenerateENO := "TRUE" } Move(in := #VeloLentaUp_Garras, out1 => #ConsignaFR_Garras)
   END_RUNG
   // the same network as SCL:
   // ENO of a box is taken as its EN; it also drops when the box reports an error
   #_w1 := NOT #EstadoZona.Manual_CBx;
   #_w2 := #_w1 AND #DestinoGarra_DOWN;
   IF #_w2 THEN #ConsignaFR_Garras := #VeloRapidaDown_Garras; END_IF;
   IF #_w2 AND #MoverGarra_LentaDOWN THEN #ConsignaFR_Garras := #VeloLentaDown_Garras; END_IF;
   #_w3 := #_w1 AND #DestinoGarra_UP;
   IF #_w3 THEN #ConsignaFR_Garras := #VeloRapidaUp_Garras; END_IF;
   IF #_w3 AND #MoverGarra_LentaUP THEN #ConsignaFR_Garras := #VeloLentaUp_Garras; END_IF;
END_REGION

REGION Network 49: --- Variador
   RUNG wire#powerrail
      Contact( #MoverGarras )
      Contact( #EstadoZona.Marcha_CBx )
      I_Contact( #EstadoZona.Error_CBx )
      I_Contact( #Error_Tx )
      { S7_Templates := "time_type := Time" } #TEsperaMoverGarras.TON(pt := t#500ms, et =>)
   END_RUNG
   // the same network as SCL:
   #TEsperaMoverGarras(IN := #MoverGarras AND #EstadoZona.Marcha_CBx AND NOT #EstadoZona.Error_CBx AND NOT #Error_Tx,   // TON
                       PT := t#500ms);
END_REGION

REGION Network 50: ----
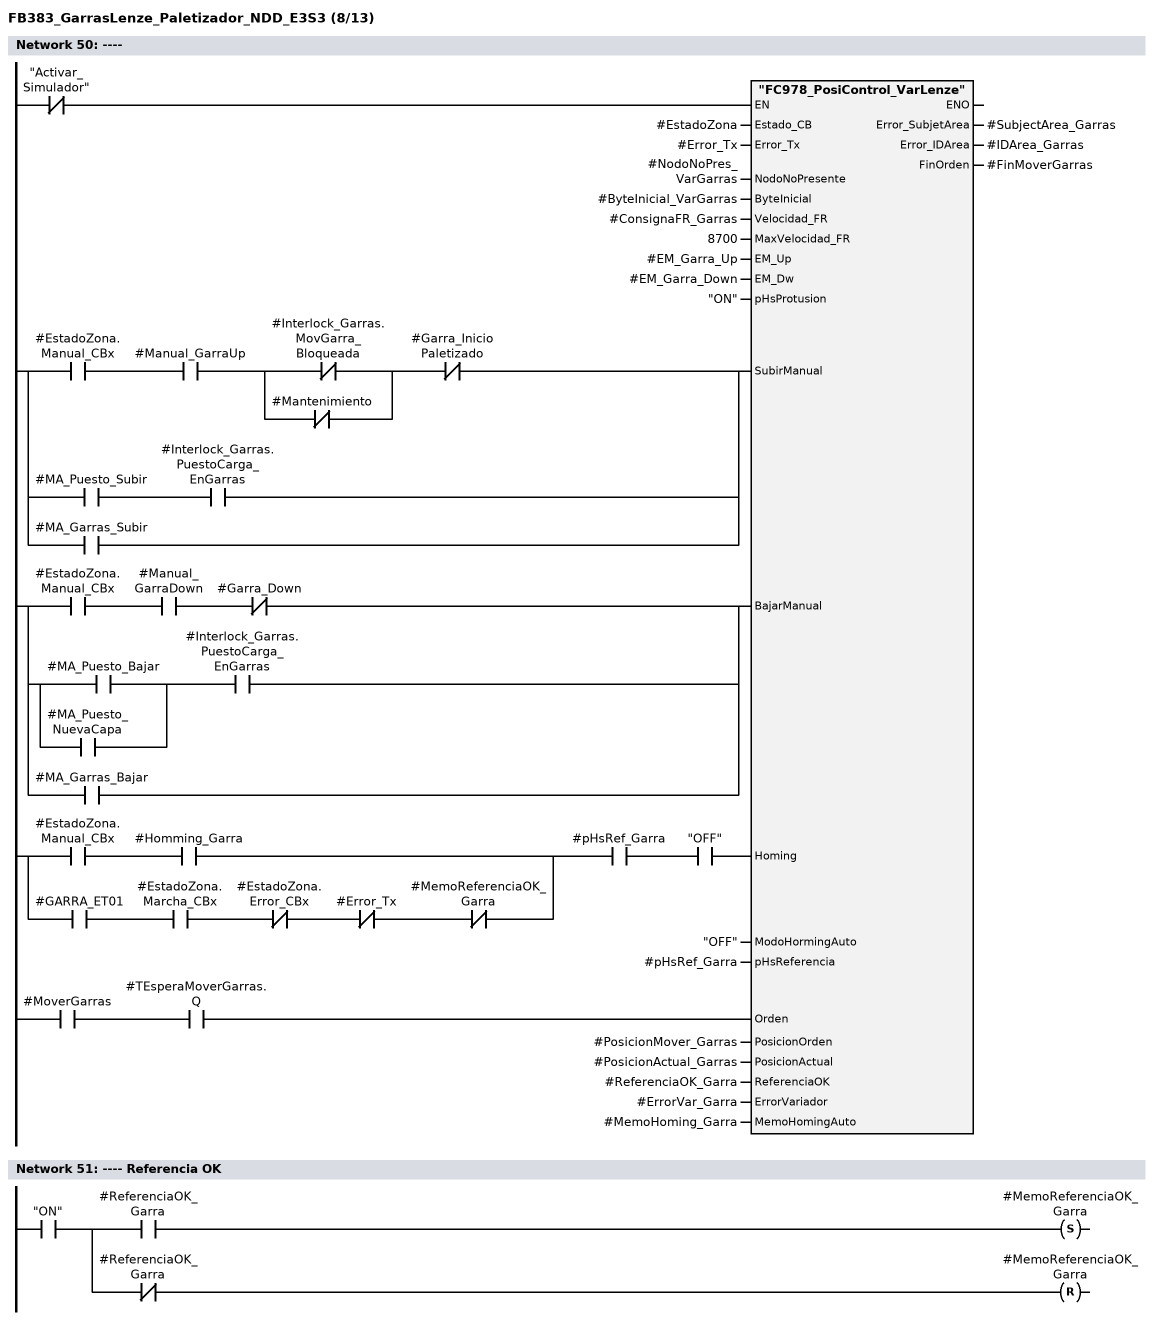
   RUNG wire#powerrail
      I_Contact( "Activar_Simulador" )
      "FC978_PosiControl_VarLenze"(SubirManual := wire#w3, BajarManual := wire#w5, Homing := wire#w7, Orden := wire#w8, Estado_CB := #EstadoZona, Error_Tx := #Error_Tx, NodoNoPresente := #NodoNoPres_VarGarras, ByteInicial := #ByteInicial_VarGarras, Velocidad_FR := #ConsignaFR_Garras, MaxVelocidad_FR := 8700, EM_Up := #EM_Garra_Up, EM_Dw := #EM_Garra_Down, pHsProtusion := "ON", ModoHormingAuto := "OFF", pHsReferencia := #pHsRef_Garra, PosicionOrden := #PosicionMover_Garras, PosicionActual := #PosicionActual_Garras, ReferenciaOK := #ReferenciaOK_Garra, ErrorVariador := #ErrorVar_Garra, MemoHomingAuto := #MemoHoming_Garra, Error_SubjetArea => #SubjectArea_Garras, Error_IDArea => #IDArea_Garras, FinOrden => #FinMoverGarras)
   END_RUNG
   RUNG wire#powerrail
      Contact( #EstadoZona.Manual_CBx )
      Contact( #Manual_GarraUp )
      wire#w1
      I_Contact( #Interlock_Garras.MovGarra_Bloqueada )
      wire#w2
      I_Contact( #Garra_InicioPaletizado )
   END_RUNG wire#w3
   RUNG wire#w1
      I_Contact( #Mantenimiento )
   END_RUNG wire#w2
   RUNG wire#powerrail
      Contact( #MA_Puesto_Subir )
      Contact( #Interlock_Garras.PuestoCarga_EnGarras )
   END_RUNG wire#w3
   RUNG wire#powerrail
      Contact( #MA_Garras_Subir )
   END_RUNG wire#w3
   RUNG wire#powerrail
      Contact( #EstadoZona.Manual_CBx )
      Contact( #Manual_GarraDown )
      I_Contact( #Garra_Down )
   END_RUNG wire#w5
   RUNG wire#powerrail
      Contact( #MA_Puesto_Bajar )
      wire#w4
      Contact( #Interlock_Garras.PuestoCarga_EnGarras )
   END_RUNG wire#w5
   RUNG wire#powerrail
      Contact( #MA_Puesto_NuevaCapa )
   END_RUNG wire#w4
   RUNG wire#powerrail
      Contact( #MA_Garras_Bajar )
   END_RUNG wire#w5
   RUNG wire#powerrail
      Contact( #EstadoZona.Manual_CBx )
      Contact( #Homming_Garra )
      wire#w6
      Contact( #pHsRef_Garra )
      Contact( "OFF" )
   END_RUNG wire#w7
   RUNG wire#powerrail
      Contact( #GARRA_ET01 )
      Contact( #EstadoZona.Marcha_CBx )
      I_Contact( #EstadoZona.Error_CBx )
      I_Contact( #Error_Tx )
      I_Contact( #MemoReferenciaOK_Garra )
   END_RUNG wire#w6
   RUNG wire#powerrail
      Contact( #MoverGarras )
      Contact( #TEsperaMoverGarras.Q )
   END_RUNG wire#w8
   // the same network as SCL:
   IF NOT "Activar_Simulador" THEN
       "FC978_PosiControl_VarLenze"(Estado_CB := #EstadoZona,
                               Error_Tx := #Error_Tx,
                               NodoNoPresente := #NodoNoPres_VarGarras,
                               ByteInicial := #ByteInicial_VarGarras,
                               Velocidad_FR := #ConsignaFR_Garras,
                               MaxVelocidad_FR := 8700,
                               EM_Up := #EM_Garra_Up,
                               EM_Dw := #EM_Garra_Down,
                               pHsProtusion := "ON",
                               SubirManual := (#EstadoZona.Manual_CBx AND #Manual_GarraUp AND (NOT #Interlock_Garras.MovGarra_Bloqueada OR NOT #Mantenimiento) AND NOT #Garra_InicioPaletizado) OR (#MA_Puesto_Subir AND #Interlock_Garras.PuestoCarga_EnGarras) OR #MA_Garras_Subir,
                               BajarManual := (#EstadoZona.Manual_CBx AND #Manual_GarraDown AND NOT #Garra_Down) OR ((#MA_Puesto_Bajar OR #MA_Puesto_NuevaCapa) AND #Interlock_Garras.PuestoCarga_EnGarras) OR #MA_Garras_Bajar,
                               Homing := ((#EstadoZona.Manual_CBx AND #Homming_Garra) OR (#GARRA_ET01 AND #EstadoZona.Marcha_CBx AND NOT #EstadoZona.Error_CBx AND NOT #Error_Tx AND NOT #MemoReferenciaOK_Garra)) AND #pHsRef_Garra AND "OFF",
                               ModoHormingAuto := "OFF",
                               pHsReferencia := #pHsRef_Garra,
                               Orden := #MoverGarras AND #TEsperaMoverGarras.Q,
                               PosicionOrden := #PosicionMover_Garras,
                               PosicionActual := #PosicionActual_Garras,
                               ReferenciaOK := #ReferenciaOK_Garra,
                               ErrorVariador := #ErrorVar_Garra,
                               MemoHomingAuto := #MemoHoming_Garra,
                               Error_SubjetArea => #SubjectArea_Garras,
                               Error_IDArea => #IDArea_Garras,
                               FinOrden => #FinMoverGarras);
   END_IF;
END_REGION

REGION Network 51: ---- Referencia OK
   RUNG wire#powerrail
      Contact( "ON" )
      wire#w1
      Contact( #ReferenciaOK_Garra )
      S_Coil( #MemoReferenciaOK_Garra )
   END_RUNG
   RUNG wire#w1
      I_Contact( #ReferenciaOK_Garra )
      R_Coil( #MemoReferenciaOK_Garra )
   END_RUNG
   // the same network as SCL:
   IF "ON" AND #ReferenciaOK_Garra THEN #MemoReferenciaOK_Garra := TRUE; END_IF;
   IF "ON" AND NOT #ReferenciaOK_Garra THEN #MemoReferenciaOK_Garra := FALSE; END_IF;
END_REGION

REGION Network 52: Eventos de Paletizado: Inicio
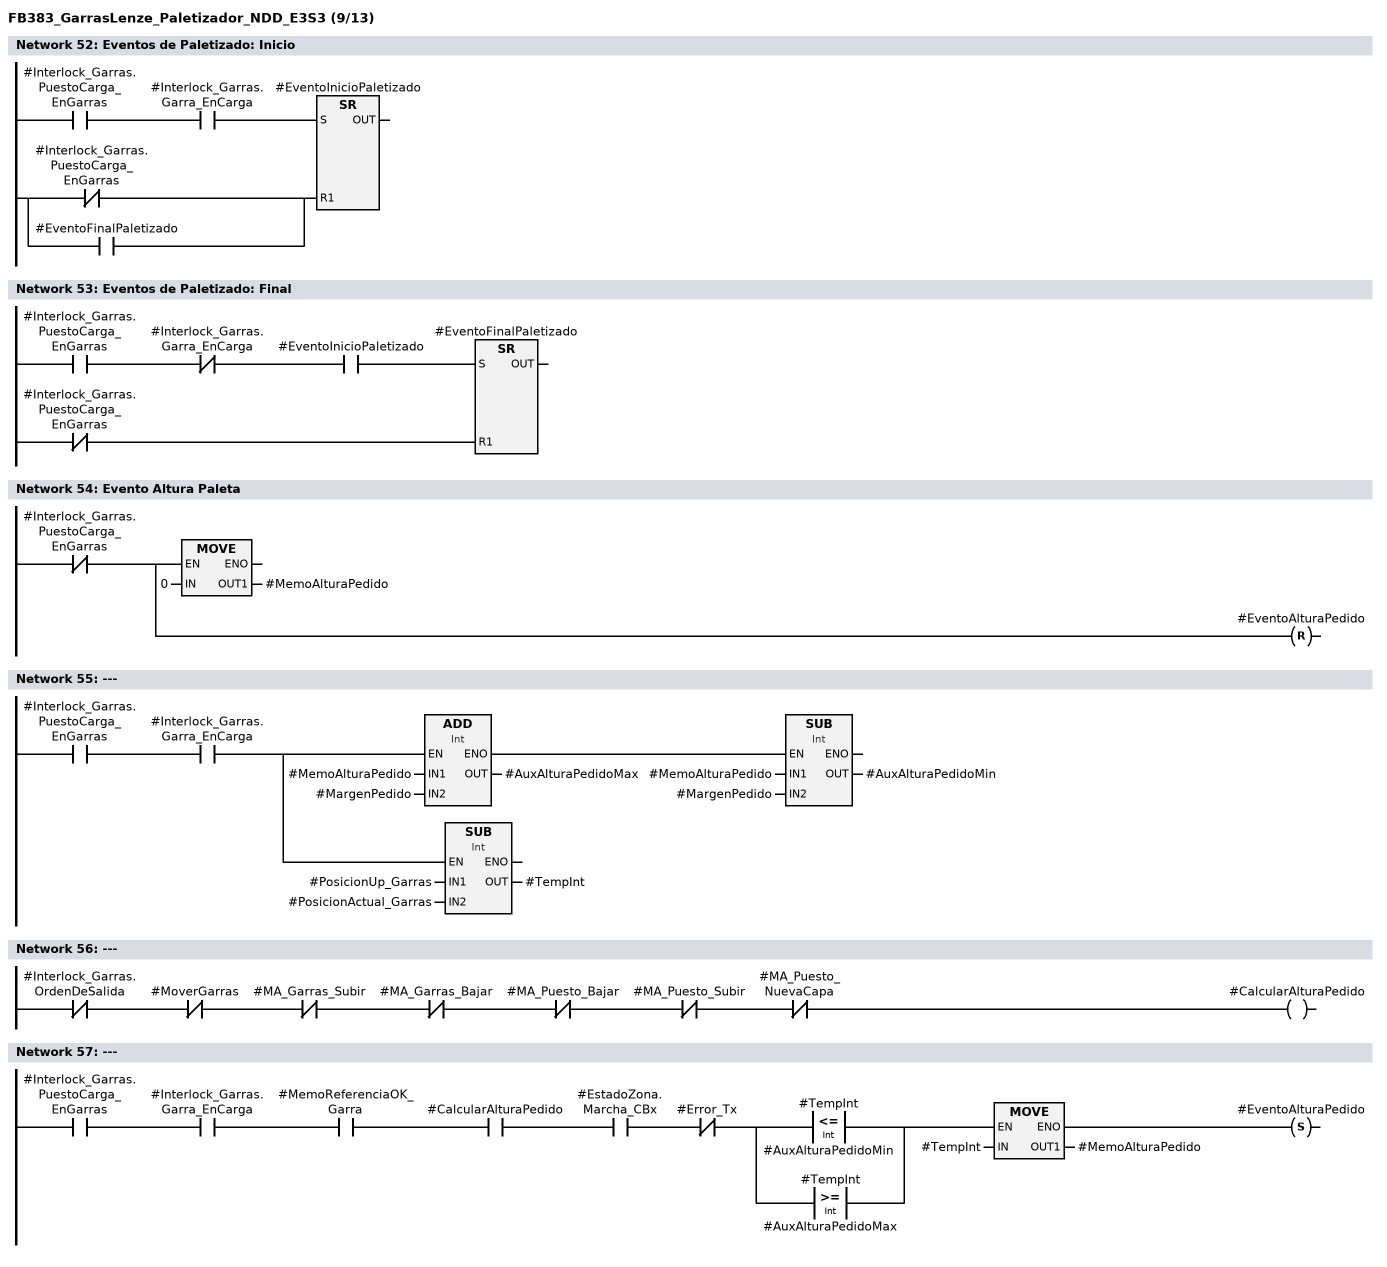
   RUNG wire#powerrail
      Contact( #Interlock_Garras.PuestoCarga_EnGarras )
      Contact( #Interlock_Garras.Garra_EnCarga )
      S_SR(operand := #EventoInicioPaletizado, r1 := wire#w1)
   END_RUNG
   RUNG wire#powerrail
      I_Contact( #Interlock_Garras.PuestoCarga_EnGarras )
   END_RUNG wire#w1
   RUNG wire#powerrail
      Contact( #EventoFinalPaletizado )
   END_RUNG wire#w1
   // the same network as SCL:
   IF #Interlock_Garras.PuestoCarga_EnGarras AND #Interlock_Garras.Garra_EnCarga THEN
       #EventoInicioPaletizado := TRUE;   // SR flip-flop
   END_IF;
   IF NOT #Interlock_Garras.PuestoCarga_EnGarras OR #EventoFinalPaletizado THEN
       #EventoInicioPaletizado := FALSE;
   END_IF;
END_REGION

REGION Network 53: Eventos de Paletizado: Final
   RUNG wire#powerrail
      Contact( #Interlock_Garras.PuestoCarga_EnGarras )
      I_Contact( #Interlock_Garras.Garra_EnCarga )
      Contact( #EventoInicioPaletizado )
      S_SR(operand := #EventoFinalPaletizado, r1 := wire#w1)
   END_RUNG
   RUNG wire#powerrail
      I_Contact( #Interlock_Garras.PuestoCarga_EnGarras )
   END_RUNG wire#w1
   // the same network as SCL:
   IF #Interlock_Garras.PuestoCarga_EnGarras AND NOT #Interlock_Garras.Garra_EnCarga AND #EventoInicioPaletizado THEN
       #EventoFinalPaletizado := TRUE;   // SR flip-flop
   END_IF;
   IF NOT #Interlock_Garras.PuestoCarga_EnGarras THEN #EventoFinalPaletizado := FALSE; END_IF;
END_REGION

REGION Network 54: Evento Altura Paleta
   RUNG wire#powerrail
      I_Contact( #Interlock_Garras.PuestoCarga_EnGarras )
      wire#w1
      { S7_GenerateENO := "TRUE" } Move(in := 0, out1 => #MemoAlturaPedido)
   END_RUNG
   RUNG wire#w1
      R_Coil( #EventoAlturaPedido )
   END_RUNG
   // the same network as SCL:
   IF NOT #Interlock_Garras.PuestoCarga_EnGarras THEN
       #MemoAlturaPedido := 0;
       #EventoAlturaPedido := FALSE;
   END_IF;
END_REGION

REGION Network 55: ---
   RUNG wire#powerrail
      Contact( #Interlock_Garras.PuestoCarga_EnGarras )
      Contact( #Interlock_Garras.Garra_EnCarga )
      wire#w1
      { S7_Templates := "SrcType := Int"; S7_GenerateENO := "TRUE" } Add(in1 := #MemoAlturaPedido, in2 := #MargenPedido, out => #AuxAlturaPedidoMax)
      { S7_Templates := "SrcType := Int"; S7_GenerateENO := "TRUE" } Sub(in1 := #MemoAlturaPedido, in2 := #MargenPedido, out => #AuxAlturaPedidoMin)
   END_RUNG
   RUNG wire#w1
      { S7_Templates := "SrcType := Int"; S7_GenerateENO := "TRUE" } Sub(in1 := #PosicionUp_Garras, in2 := #PosicionActual_Garras, out => #TempInt)
   END_RUNG
   // the same network as SCL:
   // ENO of a box is taken as its EN; it also drops when the box reports an error
   IF #Interlock_Garras.PuestoCarga_EnGarras AND #Interlock_Garras.Garra_EnCarga THEN
       #AuxAlturaPedidoMax := #MemoAlturaPedido + #MargenPedido;
       #AuxAlturaPedidoMin := #MemoAlturaPedido - #MargenPedido;
       #TempInt := #PosicionUp_Garras - #PosicionActual_Garras;
   END_IF;
END_REGION

REGION Network 56: ---
   RUNG wire#powerrail
      I_Contact( #Interlock_Garras.OrdenDeSalida )
      I_Contact( #MoverGarras )
      I_Contact( #MA_Garras_Subir )
      I_Contact( #MA_Garras_Bajar )
      I_Contact( #MA_Puesto_Bajar )
      I_Contact( #MA_Puesto_Subir )
      I_Contact( #MA_Puesto_NuevaCapa )
      Coil( #CalcularAlturaPedido )
   END_RUNG
   // the same network as SCL:
   #CalcularAlturaPedido := NOT #Interlock_Garras.OrdenDeSalida AND NOT #MoverGarras AND NOT #MA_Garras_Subir AND NOT #MA_Garras_Bajar AND NOT #MA_Puesto_Bajar AND NOT #MA_Puesto_Subir AND NOT #MA_Puesto_NuevaCapa;
END_REGION

REGION Network 57: ---
   RUNG wire#powerrail
      Contact( #Interlock_Garras.PuestoCarga_EnGarras )
      Contact( #Interlock_Garras.Garra_EnCarga )
      Contact( #MemoReferenciaOK_Garra )
      Contact( #CalcularAlturaPedido )
      Contact( #EstadoZona.Marcha_CBx )
      I_Contact( #Error_Tx )
      wire#w1
      { S7_Templates := "SrcType := Int" } LE_Contact(in1 := #TempInt, in2 := #AuxAlturaPedidoMin)
      wire#w2
      { S7_GenerateENO := "TRUE" } Move(in := #TempInt, out1 => #MemoAlturaPedido)
      S_Coil( #EventoAlturaPedido )
   END_RUNG
   RUNG wire#w1
      { S7_Templates := "SrcType := Int" } GE_Contact(in1 := #TempInt, in2 := #AuxAlturaPedidoMax)
   END_RUNG wire#w2
   // the same network as SCL:
   // ENO of a box is taken as its EN; it also drops when the box reports an error
   IF #Interlock_Garras.PuestoCarga_EnGarras AND #Interlock_Garras.Garra_EnCarga AND #MemoReferenciaOK_Garra AND #CalcularAlturaPedido AND #EstadoZona.Marcha_CBx AND NOT #Error_Tx AND ((#TempInt <= #AuxAlturaPedidoMin) OR (#TempInt >= #AuxAlturaPedidoMax)) THEN
       #MemoAlturaPedido := #TempInt;
       #EventoAlturaPedido := TRUE;
   END_IF;
END_REGION

REGION Network 58: ---
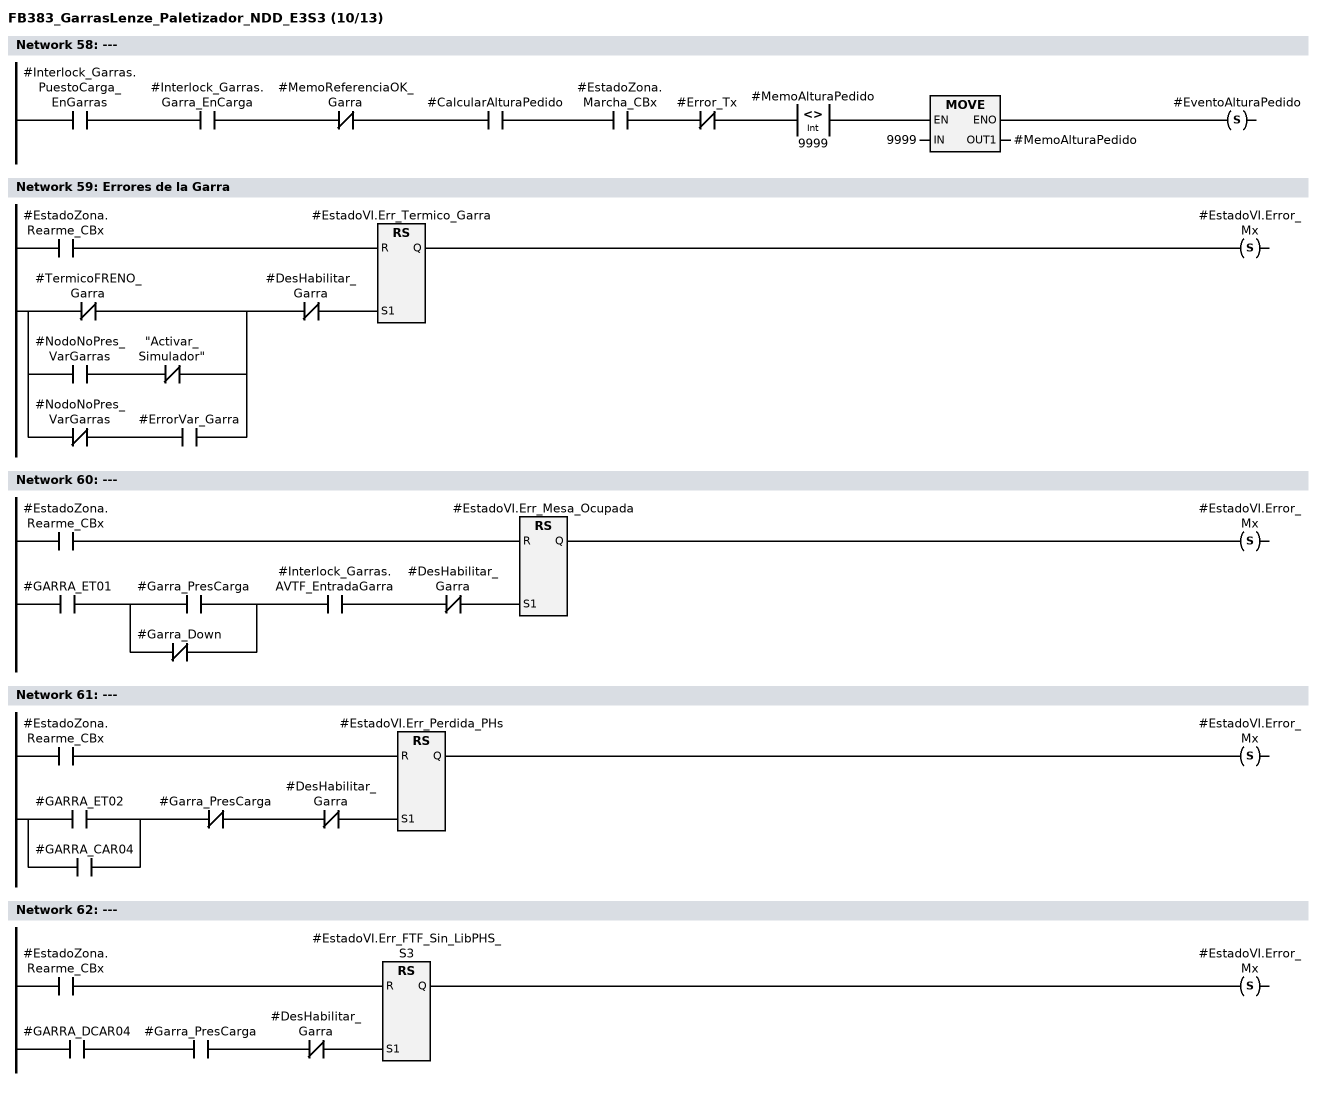
   RUNG wire#powerrail
      Contact( #Interlock_Garras.PuestoCarga_EnGarras )
      Contact( #Interlock_Garras.Garra_EnCarga )
      I_Contact( #MemoReferenciaOK_Garra )
      Contact( #CalcularAlturaPedido )
      Contact( #EstadoZona.Marcha_CBx )
      I_Contact( #Error_Tx )
      { S7_Templates := "SrcType := Int" } NE_Contact(in1 := #MemoAlturaPedido, in2 := 9999)
      { S7_GenerateENO := "TRUE" } Move(in := 9999, out1 => #MemoAlturaPedido)
      S_Coil( #EventoAlturaPedido )
   END_RUNG
   // the same network as SCL:
   // ENO of a box is taken as its EN; it also drops when the box reports an error
   #_w1 := #Interlock_Garras.PuestoCarga_EnGarras AND #Interlock_Garras.Garra_EnCarga AND NOT #MemoReferenciaOK_Garra AND #CalcularAlturaPedido AND #EstadoZona.Marcha_CBx AND NOT #Error_Tx AND (#MemoAlturaPedido <> 9999);
   IF #_w1 THEN
       #MemoAlturaPedido := 9999;
       #EventoAlturaPedido := TRUE;
   END_IF;
END_REGION

REGION Network 59: Errores de la Garra
   RUNG wire#powerrail
      Contact( #EstadoZona.Rearme_CBx )
      S_RS(operand := #EstadoVI.Err_Termico_Garra, s1 := wire#w2)
      S_Coil( #EstadoVI.Error_Mx )
   END_RUNG
   RUNG wire#powerrail
      I_Contact( #TermicoFRENO_Garra )
      wire#w1
      I_Contact( #DesHabilitar_Garra )
   END_RUNG wire#w2
   RUNG wire#powerrail
      Contact( #NodoNoPres_VarGarras )
      I_Contact( "Activar_Simulador" )
   END_RUNG wire#w1
   RUNG wire#powerrail
      I_Contact( #NodoNoPres_VarGarras )
      Contact( #ErrorVar_Garra )
   END_RUNG wire#w1
   // the same network as SCL:
   IF #EstadoZona.Rearme_CBx THEN
       #EstadoVI.Err_Termico_Garra := FALSE;   // RS flip-flop
   END_IF;
   IF (NOT #TermicoFRENO_Garra OR (#NodoNoPres_VarGarras AND NOT "Activar_Simulador") OR (NOT #NodoNoPres_VarGarras AND #ErrorVar_Garra)) AND NOT #DesHabilitar_Garra THEN
       #EstadoVI.Err_Termico_Garra := TRUE;
   END_IF;
   IF #EstadoVI.Err_Termico_Garra THEN #EstadoVI.Error_Mx := TRUE; END_IF;
END_REGION

REGION Network 60: ---
   RUNG wire#powerrail
      Contact( #EstadoZona.Rearme_CBx )
      S_RS(operand := #EstadoVI.Err_Mesa_Ocupada, s1 := wire#w3)
      S_Coil( #EstadoVI.Error_Mx )
   END_RUNG
   RUNG wire#powerrail
      Contact( #GARRA_ET01 )
      wire#w1
      Contact( #Garra_PresCarga )
      wire#w2
      Contact( #Interlock_Garras.AVTF_EntradaGarra )
      I_Contact( #DesHabilitar_Garra )
   END_RUNG wire#w3
   RUNG wire#w1
      I_Contact( #Garra_Down )
   END_RUNG wire#w2
   // the same network as SCL:
   IF #EstadoZona.Rearme_CBx THEN
       #EstadoVI.Err_Mesa_Ocupada := FALSE;   // RS flip-flop
   END_IF;
   IF #GARRA_ET01 AND (#Garra_PresCarga OR NOT #Garra_Down) AND #Interlock_Garras.AVTF_EntradaGarra AND NOT #DesHabilitar_Garra THEN
       #EstadoVI.Err_Mesa_Ocupada := TRUE;
   END_IF;
   IF #EstadoVI.Err_Mesa_Ocupada THEN #EstadoVI.Error_Mx := TRUE; END_IF;
END_REGION

REGION Network 61: ---
   RUNG wire#powerrail
      Contact( #EstadoZona.Rearme_CBx )
      S_RS(operand := #EstadoVI.Err_Perdida_PHs, s1 := wire#w2)
      S_Coil( #EstadoVI.Error_Mx )
   END_RUNG
   RUNG wire#powerrail
      Contact( #GARRA_ET02 )
      wire#w1
      I_Contact( #Garra_PresCarga )
      I_Contact( #DesHabilitar_Garra )
   END_RUNG wire#w2
   RUNG wire#powerrail
      Contact( #GARRA_CAR04 )
   END_RUNG wire#w1
   // the same network as SCL:
   IF #EstadoZona.Rearme_CBx THEN
       #EstadoVI.Err_Perdida_PHs := FALSE;   // RS flip-flop
   END_IF;
   IF (#GARRA_ET02 OR #GARRA_CAR04) AND NOT #Garra_PresCarga AND NOT #DesHabilitar_Garra THEN
       #EstadoVI.Err_Perdida_PHs := TRUE;
   END_IF;
   IF #EstadoVI.Err_Perdida_PHs THEN #EstadoVI.Error_Mx := TRUE; END_IF;
END_REGION

REGION Network 62: ---
   RUNG wire#powerrail
      Contact( #EstadoZona.Rearme_CBx )
      S_RS(operand := #EstadoVI.Err_FTF_Sin_LibPHS_S3, s1 := wire#w1)
      S_Coil( #EstadoVI.Error_Mx )
   END_RUNG
   RUNG wire#powerrail
      Contact( #GARRA_DCAR04 )
      Contact( #Garra_PresCarga )
      I_Contact( #DesHabilitar_Garra )
   END_RUNG wire#w1
   // the same network as SCL:
   IF #EstadoZona.Rearme_CBx THEN
       #EstadoVI.Err_FTF_Sin_LibPHS_S3 := FALSE;   // RS flip-flop
   END_IF;
   IF #GARRA_DCAR04 AND #Garra_PresCarga AND NOT #DesHabilitar_Garra THEN
       #EstadoVI.Err_FTF_Sin_LibPHS_S3 := TRUE;
   END_IF;
   IF #EstadoVI.Err_FTF_Sin_LibPHS_S3 THEN #EstadoVI.Error_Mx := TRUE; END_IF;
END_REGION

REGION Network 63: ---
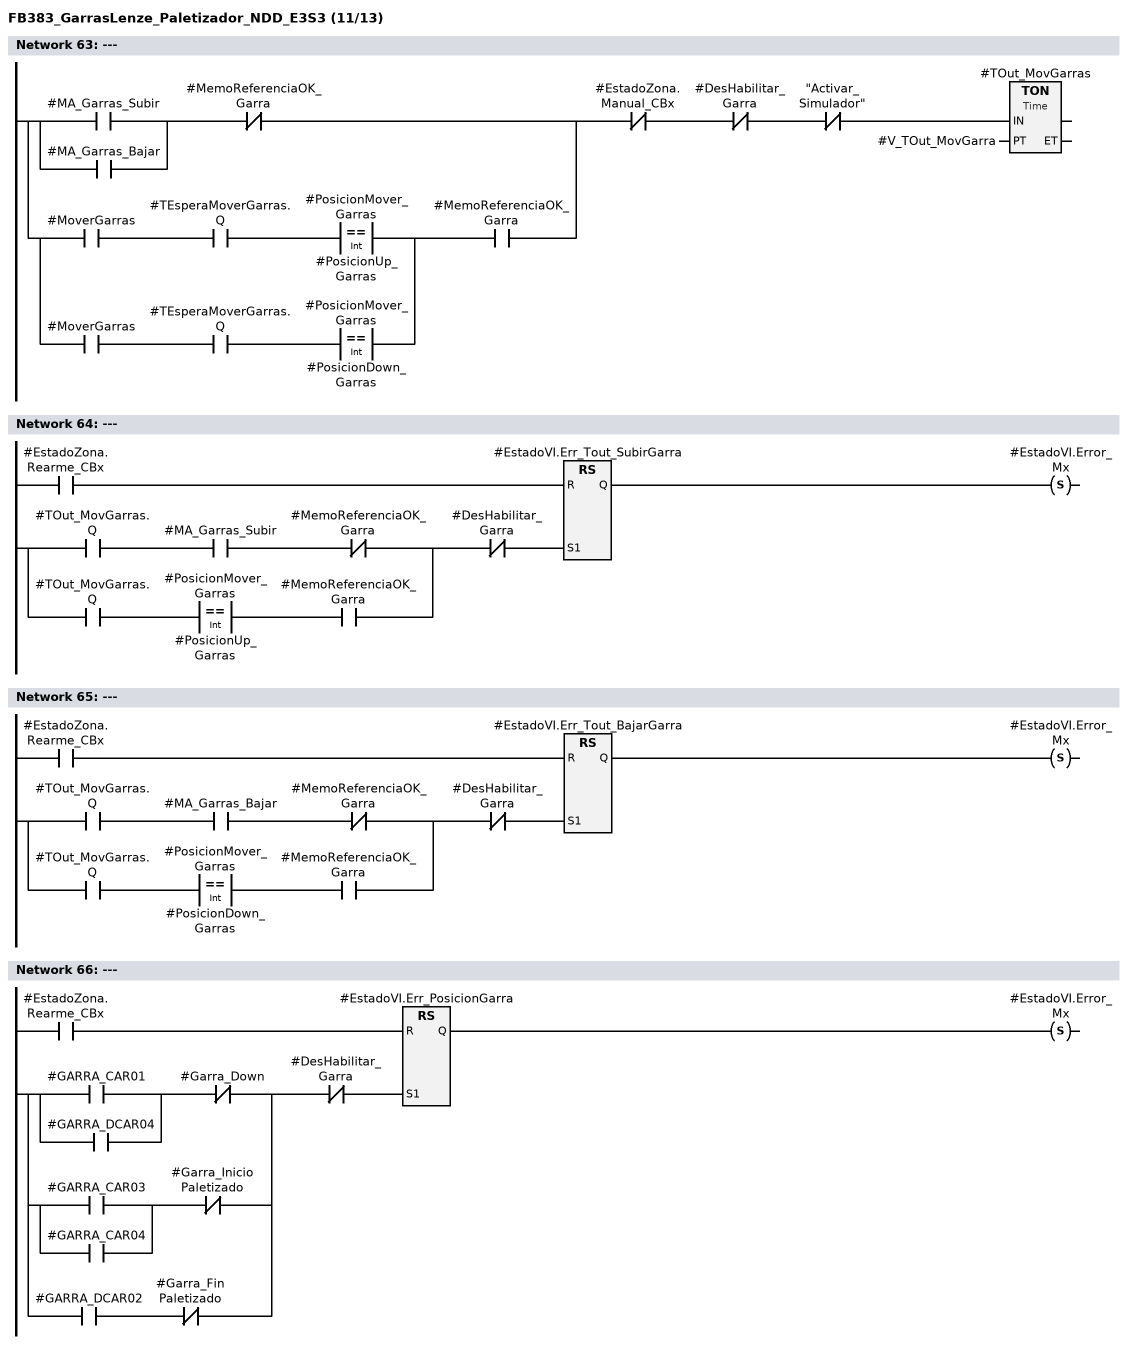
   RUNG wire#powerrail
      Contact( #MA_Garras_Subir )
      wire#w1
      I_Contact( #MemoReferenciaOK_Garra )
      wire#w2
      I_Contact( #EstadoZona.Manual_CBx )
      I_Contact( #DesHabilitar_Garra )
      I_Contact( "Activar_Simulador" )
      { S7_Templates := "time_type := Time" } #TOut_MovGarras.TON(pt := #V_TOut_MovGarra, et =>)
   END_RUNG
   RUNG wire#powerrail
      Contact( #MA_Garras_Bajar )
   END_RUNG wire#w1
   RUNG wire#powerrail
      Contact( #MoverGarras )
      Contact( #TEsperaMoverGarras.Q )
      { S7_Templates := "SrcType := Int" } EQ_Contact(in1 := #PosicionMover_Garras, in2 := #PosicionUp_Garras)
      wire#w3
      Contact( #MemoReferenciaOK_Garra )
   END_RUNG wire#w2
   RUNG wire#powerrail
      Contact( #MoverGarras )
      Contact( #TEsperaMoverGarras.Q )
      { S7_Templates := "SrcType := Int" } EQ_Contact(in1 := #PosicionMover_Garras, in2 := #PosicionDown_Garras)
   END_RUNG wire#w3
   // the same network as SCL:
   #TOut_MovGarras(IN := (((#MA_Garras_Subir OR #MA_Garras_Bajar) AND NOT #MemoReferenciaOK_Garra) OR (((#MoverGarras AND #TEsperaMoverGarras.Q AND (#PosicionMover_Garras = #PosicionUp_Garras)) OR (#MoverGarras AND #TEsperaMoverGarras.Q AND (#PosicionMover_Garras = #PosicionDown_Garras))) AND #MemoReferenciaOK_Garra)) AND NOT #EstadoZona.Manual_CBx AND NOT #DesHabilitar_Garra AND NOT "Activar_Simulador",   // TON
                   PT := #V_TOut_MovGarra);
END_REGION

REGION Network 64: ---
   RUNG wire#powerrail
      Contact( #EstadoZona.Rearme_CBx )
      S_RS(operand := #EstadoVI.Err_Tout_SubirGarra, s1 := wire#w2)
      S_Coil( #EstadoVI.Error_Mx )
   END_RUNG
   RUNG wire#powerrail
      Contact( #TOut_MovGarras.Q )
      Contact( #MA_Garras_Subir )
      I_Contact( #MemoReferenciaOK_Garra )
      wire#w1
      I_Contact( #DesHabilitar_Garra )
   END_RUNG wire#w2
   RUNG wire#powerrail
      Contact( #TOut_MovGarras.Q )
      { S7_Templates := "SrcType := Int" } EQ_Contact(in1 := #PosicionMover_Garras, in2 := #PosicionUp_Garras)
      Contact( #MemoReferenciaOK_Garra )
   END_RUNG wire#w1
   // the same network as SCL:
   IF #EstadoZona.Rearme_CBx THEN
       #EstadoVI.Err_Tout_SubirGarra := FALSE;   // RS flip-flop
   END_IF;
   IF ((#TOut_MovGarras.Q AND #MA_Garras_Subir AND NOT #MemoReferenciaOK_Garra) OR (#TOut_MovGarras.Q AND (#PosicionMover_Garras = #PosicionUp_Garras) AND #MemoReferenciaOK_Garra)) AND NOT #DesHabilitar_Garra THEN
       #EstadoVI.Err_Tout_SubirGarra := TRUE;
   END_IF;
   IF #EstadoVI.Err_Tout_SubirGarra THEN #EstadoVI.Error_Mx := TRUE; END_IF;
END_REGION

REGION Network 65: ---
   RUNG wire#powerrail
      Contact( #EstadoZona.Rearme_CBx )
      S_RS(operand := #EstadoVI.Err_Tout_BajarGarra, s1 := wire#w2)
      S_Coil( #EstadoVI.Error_Mx )
   END_RUNG
   RUNG wire#powerrail
      Contact( #TOut_MovGarras.Q )
      Contact( #MA_Garras_Bajar )
      I_Contact( #MemoReferenciaOK_Garra )
      wire#w1
      I_Contact( #DesHabilitar_Garra )
   END_RUNG wire#w2
   RUNG wire#powerrail
      Contact( #TOut_MovGarras.Q )
      { S7_Templates := "SrcType := Int" } EQ_Contact(in1 := #PosicionMover_Garras, in2 := #PosicionDown_Garras)
      Contact( #MemoReferenciaOK_Garra )
   END_RUNG wire#w1
   // the same network as SCL:
   IF #EstadoZona.Rearme_CBx THEN
       #EstadoVI.Err_Tout_BajarGarra := FALSE;   // RS flip-flop
   END_IF;
   IF ((#TOut_MovGarras.Q AND #MA_Garras_Bajar AND NOT #MemoReferenciaOK_Garra) OR (#TOut_MovGarras.Q AND (#PosicionMover_Garras = #PosicionDown_Garras) AND #MemoReferenciaOK_Garra)) AND NOT #DesHabilitar_Garra THEN
       #EstadoVI.Err_Tout_BajarGarra := TRUE;
   END_IF;
   IF #EstadoVI.Err_Tout_BajarGarra THEN #EstadoVI.Error_Mx := TRUE; END_IF;
END_REGION

REGION Network 66: ---
   RUNG wire#powerrail
      Contact( #EstadoZona.Rearme_CBx )
      S_RS(operand := #EstadoVI.Err_PosicionGarra, s1 := wire#w4)
      S_Coil( #EstadoVI.Error_Mx )
   END_RUNG
   RUNG wire#powerrail
      Contact( #GARRA_CAR01 )
      wire#w1
      I_Contact( #Garra_Down )
      wire#w2
      I_Contact( #DesHabilitar_Garra )
   END_RUNG wire#w4
   RUNG wire#powerrail
      Contact( #GARRA_DCAR04 )
   END_RUNG wire#w1
   RUNG wire#powerrail
      Contact( #GARRA_CAR03 )
      wire#w3
      I_Contact( #Garra_InicioPaletizado )
   END_RUNG wire#w2
   RUNG wire#powerrail
      Contact( #GARRA_CAR04 )
   END_RUNG wire#w3
   RUNG wire#powerrail
      Contact( #GARRA_DCAR02 )
      I_Contact( #Garra_FinPaletizado )
   END_RUNG wire#w2
   // the same network as SCL:
   IF #EstadoZona.Rearme_CBx THEN
       #EstadoVI.Err_PosicionGarra := FALSE;   // RS flip-flop
   END_IF;
   IF (((#GARRA_CAR01 OR #GARRA_DCAR04) AND NOT #Garra_Down) OR ((#GARRA_CAR03 OR #GARRA_CAR04) AND NOT #Garra_InicioPaletizado) OR (#GARRA_DCAR02 AND NOT #Garra_FinPaletizado)) AND NOT #DesHabilitar_Garra THEN
       #EstadoVI.Err_PosicionGarra := TRUE;
   END_IF;
   IF #EstadoVI.Err_PosicionGarra THEN #EstadoVI.Error_Mx := TRUE; END_IF;
END_REGION

REGION Network 67: ----
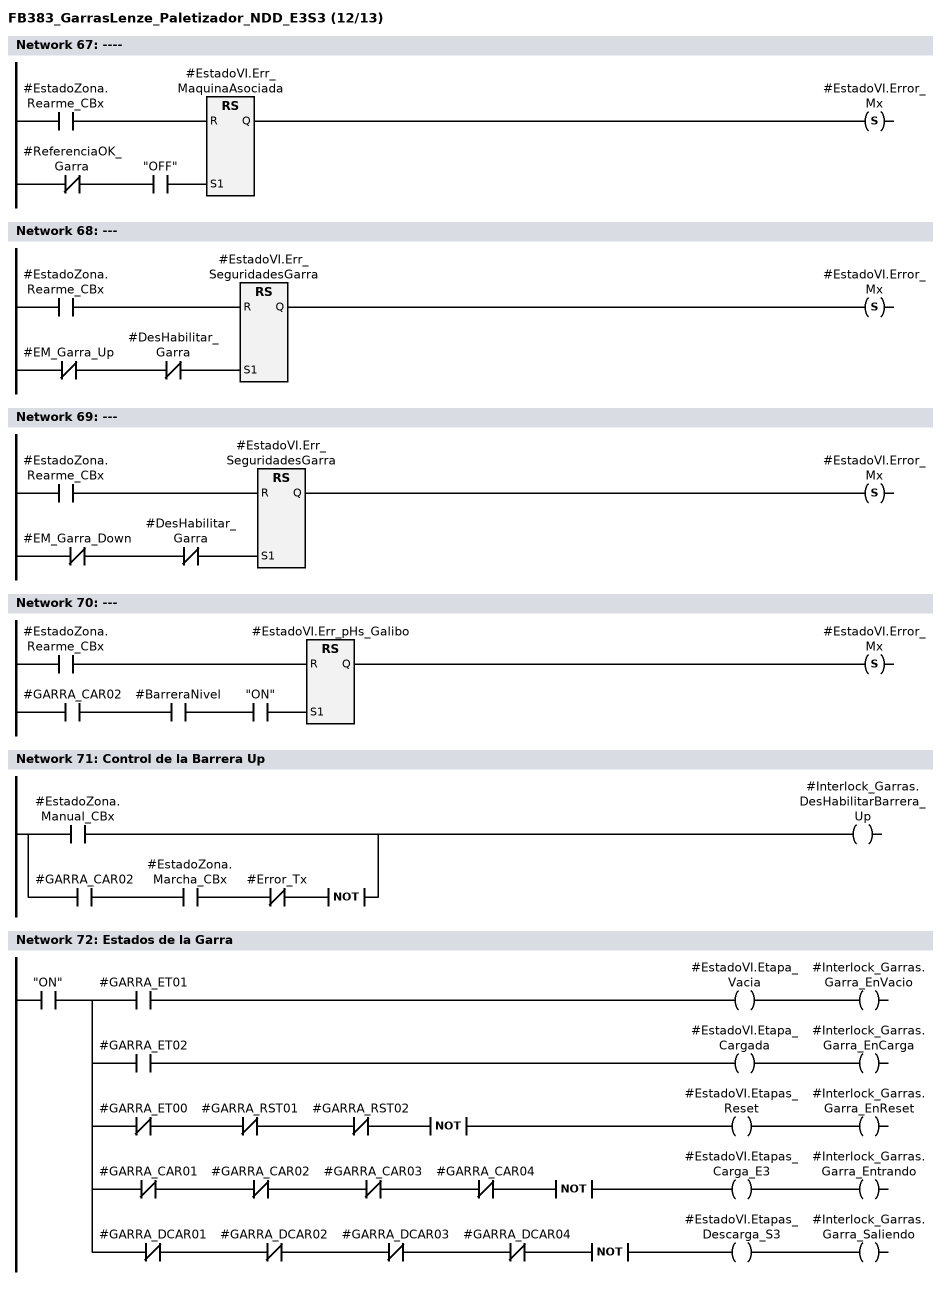
   RUNG wire#powerrail
      Contact( #EstadoZona.Rearme_CBx )
      S_RS(operand := #EstadoVI.Err_MaquinaAsociada, s1 := wire#w1)
      S_Coil( #EstadoVI.Error_Mx )
   END_RUNG
   RUNG wire#powerrail
      I_Contact( #ReferenciaOK_Garra )
      Contact( "OFF" )
   END_RUNG wire#w1
   // the same network as SCL:
   IF #EstadoZona.Rearme_CBx THEN
       #EstadoVI.Err_MaquinaAsociada := FALSE;   // RS flip-flop
   END_IF;
   IF NOT #ReferenciaOK_Garra AND "OFF" THEN #EstadoVI.Err_MaquinaAsociada := TRUE; END_IF;
   IF #EstadoVI.Err_MaquinaAsociada THEN #EstadoVI.Error_Mx := TRUE; END_IF;
END_REGION

REGION Network 68: ---
   RUNG wire#powerrail
      Contact( #EstadoZona.Rearme_CBx )
      S_RS(operand := #EstadoVI.Err_SeguridadesGarra, s1 := wire#w1)
      S_Coil( #EstadoVI.Error_Mx )
   END_RUNG
   RUNG wire#powerrail
      I_Contact( #EM_Garra_Up )
      I_Contact( #DesHabilitar_Garra )
   END_RUNG wire#w1
   // the same network as SCL:
   IF #EstadoZona.Rearme_CBx THEN
       #EstadoVI.Err_SeguridadesGarra := FALSE;   // RS flip-flop
   END_IF;
   IF NOT #EM_Garra_Up AND NOT #DesHabilitar_Garra THEN #EstadoVI.Err_SeguridadesGarra := TRUE; END_IF;
   IF #EstadoVI.Err_SeguridadesGarra THEN #EstadoVI.Error_Mx := TRUE; END_IF;
END_REGION

REGION Network 69: ---
   RUNG wire#powerrail
      Contact( #EstadoZona.Rearme_CBx )
      S_RS(operand := #EstadoVI.Err_SeguridadesGarra, s1 := wire#w1)
      S_Coil( #EstadoVI.Error_Mx )
   END_RUNG
   RUNG wire#powerrail
      I_Contact( #EM_Garra_Down )
      I_Contact( #DesHabilitar_Garra )
   END_RUNG wire#w1
   // the same network as SCL:
   IF #EstadoZona.Rearme_CBx THEN
       #EstadoVI.Err_SeguridadesGarra := FALSE;   // RS flip-flop
   END_IF;
   IF NOT #EM_Garra_Down AND NOT #DesHabilitar_Garra THEN #EstadoVI.Err_SeguridadesGarra := TRUE; END_IF;
   IF #EstadoVI.Err_SeguridadesGarra THEN #EstadoVI.Error_Mx := TRUE; END_IF;
END_REGION

REGION Network 70: ---
   RUNG wire#powerrail
      Contact( #EstadoZona.Rearme_CBx )
      S_RS(operand := #EstadoVI.Err_pHs_Galibo, s1 := wire#w1)
      S_Coil( #EstadoVI.Error_Mx )
   END_RUNG
   RUNG wire#powerrail
      Contact( #GARRA_CAR02 )
      Contact( #BarreraNivel )
      Contact( "ON" )
   END_RUNG wire#w1
   // the same network as SCL:
   IF #EstadoZona.Rearme_CBx THEN
       #EstadoVI.Err_pHs_Galibo := FALSE;   // RS flip-flop
   END_IF;
   IF #GARRA_CAR02 AND #BarreraNivel AND "ON" THEN #EstadoVI.Err_pHs_Galibo := TRUE; END_IF;
   IF #EstadoVI.Err_pHs_Galibo THEN #EstadoVI.Error_Mx := TRUE; END_IF;
END_REGION

REGION Network 71: Control de la Barrera Up
   RUNG wire#powerrail
      Contact( #EstadoZona.Manual_CBx )
      wire#w1
      Coil( #Interlock_Garras.DesHabilitarBarrera_Up )
   END_RUNG
   RUNG wire#powerrail
      Contact( #GARRA_CAR02 )
      Contact( #EstadoZona.Marcha_CBx )
      I_Contact( #Error_Tx )
      Not()
   END_RUNG wire#w1
   // the same network as SCL:
   #Interlock_Garras.DesHabilitarBarrera_Up := #EstadoZona.Manual_CBx OR NOT (#GARRA_CAR02 AND #EstadoZona.Marcha_CBx AND NOT #Error_Tx);
END_REGION

REGION Network 72: Estados de la Garra
   RUNG wire#powerrail
      Contact( "ON" )
      wire#w1
      Contact( #GARRA_ET01 )
      Coil( #EstadoVI.Etapa_Vacia )
      Coil( #Interlock_Garras.Garra_EnVacio )
   END_RUNG
   RUNG wire#w1
      Contact( #GARRA_ET02 )
      Coil( #EstadoVI.Etapa_Cargada )
      Coil( #Interlock_Garras.Garra_EnCarga )
   END_RUNG
   RUNG wire#w1
      I_Contact( #GARRA_ET00 )
      I_Contact( #GARRA_RST01 )
      I_Contact( #GARRA_RST02 )
      Not()
      Coil( #EstadoVI.Etapas_Reset )
      Coil( #Interlock_Garras.Garra_EnReset )
   END_RUNG
   RUNG wire#w1
      I_Contact( #GARRA_CAR01 )
      I_Contact( #GARRA_CAR02 )
      I_Contact( #GARRA_CAR03 )
      I_Contact( #GARRA_CAR04 )
      Not()
      Coil( #EstadoVI.Etapas_Carga_E3 )
      Coil( #Interlock_Garras.Garra_Entrando )
   END_RUNG
   RUNG wire#w1
      I_Contact( #GARRA_DCAR01 )
      I_Contact( #GARRA_DCAR02 )
      I_Contact( #GARRA_DCAR03 )
      I_Contact( #GARRA_DCAR04 )
      Not()
      Coil( #EstadoVI.Etapas_Descarga_S3 )
      Coil( #Interlock_Garras.Garra_Saliendo )
   END_RUNG
   // the same network as SCL:
   #EstadoVI.Etapa_Vacia := "ON" AND #GARRA_ET01;
   #Interlock_Garras.Garra_EnVacio := #EstadoVI.Etapa_Vacia;
   #EstadoVI.Etapa_Cargada := "ON" AND #GARRA_ET02;
   #Interlock_Garras.Garra_EnCarga := #EstadoVI.Etapa_Cargada;
   #EstadoVI.Etapas_Reset := NOT ("ON" AND NOT #GARRA_ET00 AND NOT #GARRA_RST01 AND NOT #GARRA_RST02);
   #Interlock_Garras.Garra_EnReset := #EstadoVI.Etapas_Reset;
   #EstadoVI.Etapas_Carga_E3 := NOT ("ON" AND NOT #GARRA_CAR01 AND NOT #GARRA_CAR02 AND NOT #GARRA_CAR03 AND NOT #GARRA_CAR04);
   #Interlock_Garras.Garra_Entrando := #EstadoVI.Etapas_Carga_E3;
   #EstadoVI.Etapas_Descarga_S3 := NOT ("ON" AND NOT #GARRA_DCAR01 AND NOT #GARRA_DCAR02 AND NOT #GARRA_DCAR03 AND NOT #GARRA_DCAR04);
   #Interlock_Garras.Garra_Saliendo := #EstadoVI.Etapas_Descarga_S3;
END_REGION

REGION Network 73: Entradas de la Garra
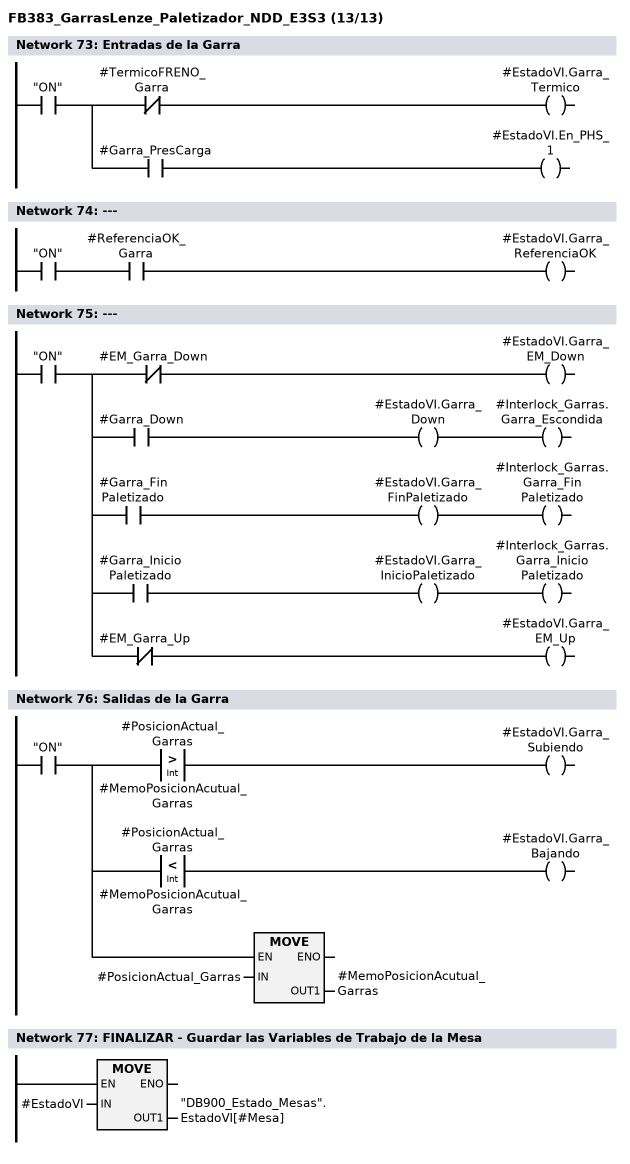
   RUNG wire#powerrail
      Contact( "ON" )
      wire#w1
      I_Contact( #TermicoFRENO_Garra )
      Coil( #EstadoVI.Garra_Termico )
   END_RUNG
   RUNG wire#w1
      Contact( #Garra_PresCarga )
      Coil( #EstadoVI.En_PHS_1 )
   END_RUNG
   // the same network as SCL:
   #EstadoVI.Garra_Termico := "ON" AND NOT #TermicoFRENO_Garra;
   #EstadoVI.En_PHS_1 := "ON" AND #Garra_PresCarga;
END_REGION

REGION Network 74: ---
   RUNG wire#powerrail
      Contact( "ON" )
      Contact( #ReferenciaOK_Garra )
      Coil( #EstadoVI.Garra_ReferenciaOK )
   END_RUNG
   // the same network as SCL:
   #EstadoVI.Garra_ReferenciaOK := "ON" AND #ReferenciaOK_Garra;
END_REGION

REGION Network 75: ---
   RUNG wire#powerrail
      Contact( "ON" )
      wire#w1
      I_Contact( #EM_Garra_Down )
      Coil( #EstadoVI.Garra_EM_Down )
   END_RUNG
   RUNG wire#w1
      Contact( #Garra_Down )
      Coil( #EstadoVI.Garra_Down )
      Coil( #Interlock_Garras.Garra_Escondida )
   END_RUNG
   RUNG wire#w1
      Contact( #Garra_FinPaletizado )
      Coil( #EstadoVI.Garra_FinPaletizado )
      Coil( #Interlock_Garras.Garra_FinPaletizado )
   END_RUNG
   RUNG wire#w1
      Contact( #Garra_InicioPaletizado )
      Coil( #EstadoVI.Garra_InicioPaletizado )
      Coil( #Interlock_Garras.Garra_InicioPaletizado )
   END_RUNG
   RUNG wire#w1
      I_Contact( #EM_Garra_Up )
      Coil( #EstadoVI.Garra_EM_Up )
   END_RUNG
   // the same network as SCL:
   #EstadoVI.Garra_EM_Down := "ON" AND NOT #EM_Garra_Down;
   #EstadoVI.Garra_Down := "ON" AND #Garra_Down;
   #Interlock_Garras.Garra_Escondida := #EstadoVI.Garra_Down;
   #EstadoVI.Garra_FinPaletizado := "ON" AND #Garra_FinPaletizado;
   #Interlock_Garras.Garra_FinPaletizado := #EstadoVI.Garra_FinPaletizado;
   #EstadoVI.Garra_InicioPaletizado := "ON" AND #Garra_InicioPaletizado;
   #Interlock_Garras.Garra_InicioPaletizado := #EstadoVI.Garra_InicioPaletizado;
   #EstadoVI.Garra_EM_Up := "ON" AND NOT #EM_Garra_Up;
END_REGION

REGION Network 76: Salidas de la Garra
   RUNG wire#powerrail
      Contact( "ON" )
      wire#w1
      { S7_Templates := "SrcType := Int" } GT_Contact(in1 := #PosicionActual_Garras, in2 := #MemoPosicionAcutual_Garras)
      Coil( #EstadoVI.Garra_Subiendo )
   END_RUNG
   RUNG wire#w1
      { S7_Templates := "SrcType := Int" } LT_Contact(in1 := #PosicionActual_Garras, in2 := #MemoPosicionAcutual_Garras)
      Coil( #EstadoVI.Garra_Bajando )
   END_RUNG
   RUNG wire#w1
      Move(in := #PosicionActual_Garras, out1 => #MemoPosicionAcutual_Garras)
   END_RUNG
   // the same network as SCL:
   #EstadoVI.Garra_Subiendo := "ON" AND (#PosicionActual_Garras > #MemoPosicionAcutual_Garras);
   #EstadoVI.Garra_Bajando := "ON" AND (#PosicionActual_Garras < #MemoPosicionAcutual_Garras);
   IF "ON" THEN #MemoPosicionAcutual_Garras := #PosicionActual_Garras; END_IF;
END_REGION

REGION Network 77: FINALIZAR - Guardar las Variables de Trabajo de la Mesa
   RUNG wire#powerrail
      Move(in := #EstadoVI, out1 => "DB900_Estado_Mesas".EstadoVI[#Mesa])
   END_RUNG
   // the same network as SCL:
   "DB900_Estado_Mesas".EstadoVI[#Mesa] := #EstadoVI;
END_REGION
END_FUNCTION_BLOCK
